temp:=Logger.s1;
ADDSTRING(ADR(tempRaw), ADR(temp), tempRawLen);

(* Sparo i COIL **)
FOR x:= 1 TO 65 DO
	temp:=CONCAT(SEL(MB_BitStatoCoil[x],'0','1'),';');
	ADDSTRING(ADR(tempRaw), ADR(temp), tempRawLen);
END_FOR

(* Sparo gli ingressi Digitali **)
FOR x:= 1 TO 358 DO
	temp:=CONCAT(SEL(MB_BitStato[x],'0','1'),';');
	ADDSTRING(ADR(tempRaw), ADR(temp), tempRawLen);
END_FOR

(* Sparo gli HOLDING **)
FOR x:= 1 TO 168 DO
	temp:=CONCAT(INT_TO_STRING(MB_RegistriHoldingLetti[x]),';');
	ADDSTRING(ADR(tempRaw), ADR(temp), tempRawLen);
END_FOR

(* Sparo gli integer **)
FOR x:= 1 TO 283 DO
	temp:=CONCAT(INT_TO_STRING(MB_RegistriLetti[x]),';');
	ADDSTRING(ADR(tempRaw), ADR(temp), tempRawLen);
END_FOR

	temp:=(INT_TO_STRING(MB_RegistriLetti[284]));
	ADDSTRING(ADR(tempRaw), ADR(temp), tempRawLen);

ADDSTRING(ADR(Logger.TData), ADR(tempRaw), Logger.TLen);
END_ACTION
ACTION Stm:
CASE state OF
	0:	(* Refresh time manager *)
		ReadTmr(IN:=NOT ReadTmr.Q);
		(*A tempo interrogo il nodo sempre che non ci sia qualcuno che lo sta interrogando in quel momento *)

		IF (ReadTmr.Q AND NodoDaInterrogareMB1=Address )OR Refresh_Now AND NOT InibiscoModbusMB1 THEN
			state := 10;
			ReadTmr.PT := T#10s;  (* moreno *)
			Refresh_Now := FALSE;
			InibiscoModbusMB1 := TRUE;
		END_IF

	(**** Leggo le Analogiche a Disposzione  ****)

	10:	(* richiedo lettura di tutti gli Input Register   *)

		Modbus.MB_Query.SlaveAddress := Address;
		Modbus.MB_Query.FunctionCode := 4;
		Read_StartAddress := 0 ;			(* richiedo lettura altri Parametri *)
		Read_Quantity := 20;
		ModBus.MB_Start := TRUE;
		state := 20;


	20:
		ModBus.MB_Query.Read_StartAddress := 0 ;			(* richiedo lettura altri Parametri *)
		ModBus.MB_Query.Read_Quantity := 20;
		ModBus.MB_Start := TRUE;
		Read_StartAddress := 0 ;
		state := 30;



	30:	(* Risposta all'interrogazione *)
		IF NOT ModBus.MB_Start   THEN
			VerificaFuctionCode:=ModBus.MB_Resp.FunctionCode;
			VerificaNodoLetto:=ModBus.MB_Resp.SlaveAddress;

			IF ModBus.MB_MASTER.MB_Error<>0 THEN
				state := 300;
			ELSE

				FOR x:= 0 TO ModBus.MB_Query.Read_Quantity DO
					MB_RegistriLetti[Read_StartAddress+x ] := ModBus.MB_Resp.Data[x];   	(* Vedi tabella *)
				END_FOR

			ModBus.MB_Query.Read_StartAddress := 20 ;			(* richiedo lettura altri Parametri *)
			ModBus.MB_Query.Read_Quantity := 20;
			ModBus.MB_Start := TRUE;
			Read_StartAddress := 20 ;
			state := 31;
			END_IF
		END_IF


	31:	(* Risposta all'interrogazione *)
		IF NOT ModBus.MB_Start   THEN
			VerificaFuctionCode:=ModBus.MB_Resp.FunctionCode;
			VerificaNodoLetto:=ModBus.MB_Resp.SlaveAddress;

			IF ModBus.MB_MASTER.MB_Error<>0 THEN
				state := 300;
			ELSE

				FOR x:= 0 TO ModBus.MB_Query.Read_Quantity DO
					MB_RegistriLetti[Read_StartAddress+x ] := ModBus.MB_Resp.Data[x];   	(* Vedi tabella *)
				END_FOR

			ModBus.MB_Query.Read_StartAddress := 40 ;			(* richiedo lettura altri Parametri *)
			ModBus.MB_Query.Read_Quantity := 20;
			ModBus.MB_Start := TRUE;
			Read_StartAddress := 40 ;
			state := 32;
			END_IF
		END_IF



	32:	(* Risposta all'interrogazione *)
		IF NOT ModBus.MB_Start   THEN
			VerificaFuctionCode:=ModBus.MB_Resp.FunctionCode;
			VerificaNodoLetto:=ModBus.MB_Resp.SlaveAddress;

			IF ModBus.MB_MASTER.MB_Error<>0 THEN
				state := 300;
			ELSE

				FOR x:= 0 TO ModBus.MB_Query.Read_Quantity DO
					MB_RegistriLetti[Read_StartAddress+x ] := ModBus.MB_Resp.Data[x];   	(* Vedi tabella *)
				END_FOR

			ModBus.MB_Query.Read_StartAddress := 60 ;			(* richiedo lettura altri Parametri *)
			ModBus.MB_Query.Read_Quantity := 20;
			ModBus.MB_Start := TRUE;
			Read_StartAddress := 60 ;
			state := 33;
			END_IF
		END_IF

	33:	(* Risposta all'interrogazione *)
		IF NOT ModBus.MB_Start   THEN
			VerificaFuctionCode:=ModBus.MB_Resp.FunctionCode;
			VerificaNodoLetto:=ModBus.MB_Resp.SlaveAddress;

			IF ModBus.MB_MASTER.MB_Error<>0 THEN
				state := 300;
			ELSE

				FOR x:= 0 TO ModBus.MB_Query.Read_Quantity DO
					MB_RegistriLetti[Read_StartAddress+x ] := ModBus.MB_Resp.Data[x];   	(* Vedi tabella *)
				END_FOR

			ModBus.MB_Query.Read_StartAddress := 80 ;			(* richiedo lettura altri Parametri *)
			ModBus.MB_Query.Read_Quantity := 20;
			ModBus.MB_Start := TRUE;
			Read_StartAddress := 80 ;
			state := 34;
			END_IF
		END_IF


	34:	(* Risposta all'interrogazione *)
		IF NOT ModBus.MB_Start   THEN
			VerificaFuctionCode:=ModBus.MB_Resp.FunctionCode;
			VerificaNodoLetto:=ModBus.MB_Resp.SlaveAddress;

			IF ModBus.MB_MASTER.MB_Error<>0 THEN
				state := 300;
			ELSE

				FOR x:= 0 TO ModBus.MB_Query.Read_Quantity DO
					MB_RegistriLetti[Read_StartAddress+x ] := ModBus.MB_Resp.Data[x];   	(* Vedi tabella *)
				END_FOR

			ModBus.MB_Query.Read_StartAddress := 100 ;			(* richiedo lettura altri Parametri *)
			ModBus.MB_Query.Read_Quantity := 20;
			ModBus.MB_Start := TRUE;
			Read_StartAddress := 100 ;
			state := 35;
			END_IF
		END_IF


	35:	(* Risposta all'interrogazione *)
		IF NOT ModBus.MB_Start   THEN
			VerificaFuctionCode:=ModBus.MB_Resp.FunctionCode;
			VerificaNodoLetto:=ModBus.MB_Resp.SlaveAddress;

			IF ModBus.MB_MASTER.MB_Error<>0 THEN
				state := 300;
			ELSE

				FOR x:= 0 TO ModBus.MB_Query.Read_Quantity DO
					MB_RegistriLetti[Read_StartAddress+x ] := ModBus.MB_Resp.Data[x];   	(* Vedi tabella *)
				END_FOR

			ModBus.MB_Query.Read_StartAddress := 120 ;			(* richiedo lettura altri Parametri *)
			ModBus.MB_Query.Read_Quantity := 20;
			ModBus.MB_Start := TRUE;
			Read_StartAddress := 120 ;
			state := 36;
			END_IF
		END_IF

	36:	(* Risposta all'interrogazione *)
		IF NOT ModBus.MB_Start   THEN
			VerificaFuctionCode:=ModBus.MB_Resp.FunctionCode;
			VerificaNodoLetto:=ModBus.MB_Resp.SlaveAddress;

			IF ModBus.MB_MASTER.MB_Error<>0 THEN
				state := 300;
			ELSE

				FOR x:= 0 TO ModBus.MB_Query.Read_Quantity DO
					MB_RegistriLetti[Read_StartAddress+x ] := ModBus.MB_Resp.Data[x];   	(* Vedi tabella *)
				END_FOR

			ModBus.MB_Query.Read_StartAddress := 140 ;			(* richiedo lettura altri Parametri *)
			ModBus.MB_Query.Read_Quantity := 20;
			ModBus.MB_Start := TRUE;
			Read_StartAddress := 140 ;
			state := 37;
			END_IF
		END_IF

	37:	(* Risposta all'interrogazione *)
		IF NOT ModBus.MB_Start   THEN
			VerificaFuctionCode:=ModBus.MB_Resp.FunctionCode;
			VerificaNodoLetto:=ModBus.MB_Resp.SlaveAddress;

			IF ModBus.MB_MASTER.MB_Error<>0 THEN
				state := 300;
			ELSE

				FOR x:= 0 TO ModBus.MB_Query.Read_Quantity DO
					MB_RegistriLetti[Read_StartAddress+x ] := ModBus.MB_Resp.Data[x];   	(* Vedi tabella *)
				END_FOR

			ModBus.MB_Query.Read_StartAddress := 160 ;			(* richiedo lettura altri Parametri *)
			ModBus.MB_Query.Read_Quantity := 20;
			ModBus.MB_Start := TRUE;
			Read_StartAddress := 160 ;
			state := 38;
			END_IF
		END_IF

	38:	(* Risposta all'interrogazione *)
		IF NOT ModBus.MB_Start   THEN
			VerificaFuctionCode:=ModBus.MB_Resp.FunctionCode;
			VerificaNodoLetto:=ModBus.MB_Resp.SlaveAddress;

			IF ModBus.MB_MASTER.MB_Error<>0 THEN
				state := 300;
			ELSE

				FOR x:= 0 TO ModBus.MB_Query.Read_Quantity DO
					MB_RegistriLetti[Read_StartAddress+x ] := ModBus.MB_Resp.Data[x];   	(* Vedi tabella *)
				END_FOR

			ModBus.MB_Query.Read_StartAddress := 180 ;			(* richiedo lettura altri Parametri *)
			ModBus.MB_Query.Read_Quantity := 20;
			ModBus.MB_Start := TRUE;
			Read_StartAddress := 180 ;
			state := 39;
			END_IF
		END_IF

	39:	(* Risposta all'interrogazione *)
		IF NOT ModBus.MB_Start   THEN
			VerificaFuctionCode:=ModBus.MB_Resp.FunctionCode;
			VerificaNodoLetto:=ModBus.MB_Resp.SlaveAddress;

			IF ModBus.MB_MASTER.MB_Error<>0 THEN
				state := 300;
			ELSE

				FOR x:= 0 TO ModBus.MB_Query.Read_Quantity DO
					MB_RegistriLetti[Read_StartAddress+x ] := ModBus.MB_Resp.Data[x];   	(* Vedi tabella *)
				END_FOR

			ModBus.MB_Query.Read_StartAddress := 200 ;			(* richiedo lettura altri Parametri *)
			ModBus.MB_Query.Read_Quantity := 20;
			ModBus.MB_Start := TRUE;
			Read_StartAddress := 200 ;
			state := 40;
			END_IF
		END_IF

	40:	(* Risposta all'interrogazione *)
		IF NOT ModBus.MB_Start   THEN
			VerificaFuctionCode:=ModBus.MB_Resp.FunctionCode;
			VerificaNodoLetto:=ModBus.MB_Resp.SlaveAddress;

			IF ModBus.MB_MASTER.MB_Error<>0 THEN
				state := 300;
			ELSE

				FOR x:= 0 TO ModBus.MB_Query.Read_Quantity DO
					MB_RegistriLetti[Read_StartAddress+x ] := ModBus.MB_Resp.Data[x];   	(* Vedi tabella *)
				END_FOR

			ModBus.MB_Query.Read_StartAddress := 220 ;			(* richiedo lettura altri Parametri *)
			ModBus.MB_Query.Read_Quantity := 20;
			ModBus.MB_Start := TRUE;
			Read_StartAddress := 220 ;
			state := 41;
			END_IF
		END_IF

	41:	(* Risposta all'interrogazione *)
		IF NOT ModBus.MB_Start   THEN
			VerificaFuctionCode:=ModBus.MB_Resp.FunctionCode;
			VerificaNodoLetto:=ModBus.MB_Resp.SlaveAddress;

			IF ModBus.MB_MASTER.MB_Error<>0 THEN
				state := 300;
			ELSE

				FOR x:= 0 TO ModBus.MB_Query.Read_Quantity DO
					MB_RegistriLetti[Read_StartAddress+x ] := ModBus.MB_Resp.Data[x];   	(* Vedi tabella *)
				END_FOR

			ModBus.MB_Query.Read_StartAddress := 240 ;			(* richiedo lettura altri Parametri *)
			ModBus.MB_Query.Read_Quantity := 20;
			ModBus.MB_Start := TRUE;
			Read_StartAddress := 240 ;
			state := 42;
			END_IF
		END_IF

	42:	(* Risposta all'interrogazione *)
		IF NOT ModBus.MB_Start   THEN
			VerificaFuctionCode:=ModBus.MB_Resp.FunctionCode;
			VerificaNodoLetto:=ModBus.MB_Resp.SlaveAddress;

			IF ModBus.MB_MASTER.MB_Error<>0 THEN
				state := 300;
			ELSE

				FOR x:= 0 TO ModBus.MB_Query.Read_Quantity DO
					MB_RegistriLetti[Read_StartAddress+x ] := ModBus.MB_Resp.Data[x];   	(* Vedi tabella *)
				END_FOR

			ModBus.MB_Query.Read_StartAddress := 260 ;			(* richiedo lettura altri Parametri *)
			ModBus.MB_Query.Read_Quantity := 20;
			ModBus.MB_Start := TRUE;
			Read_StartAddress := 260 ;
			state := 43;
			END_IF
		END_IF

	43:	(* Risposta all'interrogazione *)
		IF NOT ModBus.MB_Start   THEN
			VerificaFuctionCode:=ModBus.MB_Resp.FunctionCode;
			VerificaNodoLetto:=ModBus.MB_Resp.SlaveAddress;

			IF ModBus.MB_MASTER.MB_Error<>0 THEN
				state := 300;
			ELSE

				FOR x:= 0 TO ModBus.MB_Query.Read_Quantity DO
					MB_RegistriLetti[Read_StartAddress+x ] := ModBus.MB_Resp.Data[x];   	(* Vedi tabella *)
				END_FOR

			ModBus.MB_Query.Read_StartAddress := 280 ;			(* richiedo lettura altri Parametri *)
			ModBus.MB_Query.Read_Quantity := 4;
			ModBus.MB_Start := TRUE;
			Read_StartAddress := 280 ;
			state := 44;
			END_IF
		END_IF

	44:	(* Risposta all'interrogazione *)
		IF NOT ModBus.MB_Start   THEN
			VerificaFuctionCode:=ModBus.MB_Resp.FunctionCode;
			VerificaNodoLetto:=ModBus.MB_Resp.SlaveAddress;

			IF ModBus.MB_MASTER.MB_Error<>0 THEN
				state := 300;
			ELSE

				FOR x:= 0 TO ModBus.MB_Query.Read_Quantity DO
					MB_RegistriLetti[Read_StartAddress+x ] := ModBus.MB_Resp.Data[x];   	(* Vedi tabella *)
				END_FOR

		(*	ModBus.MB_Query.Read_StartAddress := 280 ;			(* richiedo lettura altri Parametri *)
			ModBus.MB_Query.Read_Quantity := 4;
			ModBus.MB_Start := TRUE;
			Read_StartAddress := 280 ; *)
			state := 50;
			END_IF
		END_IF





	50:	(* Risposta all'interrogazione Holding*)

		Modbus.MB_Query.FunctionCode := 3;
		Read_StartAddress := 0 ;			(* richiedo lettura altri Parametri *)
		Read_Quantity := 20;
		ModBus.MB_Start := TRUE;
		state := 51;

	51:	(* Risposta all'interrogazione *)
		IF NOT ModBus.MB_Start   THEN
			VerificaFuctionCode:=ModBus.MB_Resp.FunctionCode;
			VerificaNodoLetto:=ModBus.MB_Resp.SlaveAddress;

			IF ModBus.MB_MASTER.MB_Error<>0 THEN
				state := 300;
			ELSE

				FOR x:= 0 TO ModBus.MB_Query.Read_Quantity DO
					MB_RegistriHoldingLetti[Read_StartAddress+x ] := ModBus.MB_Resp.Data[x];   	(* Vedi tabella *)
				END_FOR

			ModBus.MB_Query.Read_StartAddress := 0 ;			(* richiedo lettura altri Parametri *)
			ModBus.MB_Query.Read_Quantity := 20;
			ModBus.MB_Start := TRUE;
			Read_StartAddress := 0 ;
			state := 511;
			END_IF
		END_IF


	511:	(* Risposta all'interrogazione *)
		IF NOT ModBus.MB_Start   THEN
			VerificaFuctionCode:=ModBus.MB_Resp.FunctionCode;
			VerificaNodoLetto:=ModBus.MB_Resp.SlaveAddress;

			IF ModBus.MB_MASTER.MB_Error<>0 THEN
				state := 300;
			ELSE

				FOR x:= 0 TO ModBus.MB_Query.Read_Quantity DO
					MB_RegistriHoldingLetti[Read_StartAddress+x ] := ModBus.MB_Resp.Data[x];   	(* Vedi tabella *)
				END_FOR

			ModBus.MB_Query.Read_StartAddress := 20 ;			(* richiedo lettura altri Parametri *)
			ModBus.MB_Query.Read_Quantity := 20;
			ModBus.MB_Start := TRUE;
			Read_StartAddress := 20 ;
			state := 52;
			END_IF
		END_IF

	52:	(* Risposta all'interrogazione *)
		IF NOT ModBus.MB_Start   THEN
			VerificaFuctionCode:=ModBus.MB_Resp.FunctionCode;
			VerificaNodoLetto:=ModBus.MB_Resp.SlaveAddress;

			IF ModBus.MB_MASTER.MB_Error<>0 THEN
				state := 300;
			ELSE

				FOR x:= 0 TO ModBus.MB_Query.Read_Quantity DO
					MB_RegistriHoldingLetti[Read_StartAddress+x ] := ModBus.MB_Resp.Data[x];   	(* Vedi tabella *)
				END_FOR

			ModBus.MB_Query.Read_StartAddress := 40 ;			(* richiedo lettura altri Parametri *)
			ModBus.MB_Query.Read_Quantity := 20;
			ModBus.MB_Start := TRUE;
			Read_StartAddress := 40 ;
			state := 53;
			END_IF
		END_IF

	53:	(* Risposta all'interrogazione *)
		IF NOT ModBus.MB_Start   THEN
			VerificaFuctionCode:=ModBus.MB_Resp.FunctionCode;
			VerificaNodoLetto:=ModBus.MB_Resp.SlaveAddress;

			IF ModBus.MB_MASTER.MB_Error<>0 THEN
				state := 300;
			ELSE

				FOR x:= 0 TO ModBus.MB_Query.Read_Quantity DO
					MB_RegistriHoldingLetti[Read_StartAddress+x ] := ModBus.MB_Resp.Data[x];   	(* Vedi tabella *)
				END_FOR

			ModBus.MB_Query.Read_StartAddress := 60 ;			(* richiedo lettura altri Parametri *)
			ModBus.MB_Query.Read_Quantity := 20;
			ModBus.MB_Start := TRUE;
			Read_StartAddress := 60 ;
			state := 54;
			END_IF
		END_IF

	54:	(* Risposta all'interrogazione *)
		IF NOT ModBus.MB_Start   THEN
			VerificaFuctionCode:=ModBus.MB_Resp.FunctionCode;
			VerificaNodoLetto:=ModBus.MB_Resp.SlaveAddress;

			IF ModBus.MB_MASTER.MB_Error<>0 THEN
				state := 300;
			ELSE

				FOR x:= 0 TO ModBus.MB_Query.Read_Quantity DO
					MB_RegistriHoldingLetti[Read_StartAddress+x ] := ModBus.MB_Resp.Data[x];   	(* Vedi tabella *)
				END_FOR

			ModBus.MB_Query.Read_StartAddress := 80 ;			(* richiedo lettura altri Parametri *)
			ModBus.MB_Query.Read_Quantity := 20;
			ModBus.MB_Start := TRUE;
			Read_StartAddress := 80 ;
			state := 55;
			END_IF
		END_IF

	55:	(* Risposta all'interrogazione *)
		IF NOT ModBus.MB_Start   THEN
			VerificaFuctionCode:=ModBus.MB_Resp.FunctionCode;
			VerificaNodoLetto:=ModBus.MB_Resp.SlaveAddress;

			IF ModBus.MB_MASTER.MB_Error<>0 THEN
				state := 300;
			ELSE

				FOR x:= 0 TO ModBus.MB_Query.Read_Quantity DO
					MB_RegistriHoldingLetti[Read_StartAddress+x ] := ModBus.MB_Resp.Data[x];   	(* Vedi tabella *)
				END_FOR

			ModBus.MB_Query.Read_StartAddress := 100 ;			(* richiedo lettura altri Parametri *)
			ModBus.MB_Query.Read_Quantity := 20;
			ModBus.MB_Start := TRUE;
			Read_StartAddress := 100 ;
			state := 56;
			END_IF
		END_IF

	56:	(* Risposta all'interrogazione *)
		IF NOT ModBus.MB_Start   THEN
			VerificaFuctionCode:=ModBus.MB_Resp.FunctionCode;
			VerificaNodoLetto:=ModBus.MB_Resp.SlaveAddress;

			IF ModBus.MB_MASTER.MB_Error<>0 THEN
				state := 300;
			ELSE

				FOR x:= 0 TO ModBus.MB_Query.Read_Quantity DO
					MB_RegistriHoldingLetti[Read_StartAddress+x ] := ModBus.MB_Resp.Data[x];   	(* Vedi tabella *)
				END_FOR

			ModBus.MB_Query.Read_StartAddress := 120 ;			(* richiedo lettura altri Parametri *)
			ModBus.MB_Query.Read_Quantity := 20;
			ModBus.MB_Start := TRUE;
			Read_StartAddress := 120 ;
			state := 57;
			END_IF
		END_IF

	57:	(* Risposta all'interrogazione *)
		IF NOT ModBus.MB_Start   THEN
			VerificaFuctionCode:=ModBus.MB_Resp.FunctionCode;
			VerificaNodoLetto:=ModBus.MB_Resp.SlaveAddress;

			IF ModBus.MB_MASTER.MB_Error<>0 THEN
				state := 300;
			ELSE

				FOR x:= 0 TO ModBus.MB_Query.Read_Quantity DO
					MB_RegistriHoldingLetti[Read_StartAddress+x ] := ModBus.MB_Resp.Data[x];   	(* Vedi tabella *)
				END_FOR

			ModBus.MB_Query.Read_StartAddress := 140 ;			(* richiedo lettura altri Parametri *)
			ModBus.MB_Query.Read_Quantity := 20;
			ModBus.MB_Start := TRUE;
			Read_StartAddress := 140 ;
			state := 58;
			END_IF
		END_IF

	58:	(* Risposta all'interrogazione *)
		IF NOT ModBus.MB_Start   THEN
			VerificaFuctionCode:=ModBus.MB_Resp.FunctionCode;
			VerificaNodoLetto:=ModBus.MB_Resp.SlaveAddress;

			IF ModBus.MB_MASTER.MB_Error<>0 THEN
				state := 300;
			ELSE

				FOR x:= 0 TO ModBus.MB_Query.Read_Quantity DO
					MB_RegistriHoldingLetti[Read_StartAddress+x ] := ModBus.MB_Resp.Data[x];   	(* Vedi tabella *)
				END_FOR

			ModBus.MB_Query.Read_StartAddress := 160 ;			(* richiedo lettura altri Parametri *)
			ModBus.MB_Query.Read_Quantity := 8;
			ModBus.MB_Start := TRUE;
			Read_StartAddress := 160 ;
			state := 59;
			END_IF
		END_IF

	59:	(* Risposta all'interrogazione *)
		IF NOT ModBus.MB_Start   THEN
			VerificaFuctionCode:=ModBus.MB_Resp.FunctionCode;
			VerificaNodoLetto:=ModBus.MB_Resp.SlaveAddress;

			IF ModBus.MB_MASTER.MB_Error<>0 THEN
				state := 300;
			ELSE

				FOR x:= 0 TO ModBus.MB_Query.Read_Quantity DO
					MB_RegistriHoldingLetti[Read_StartAddress+x ] := ModBus.MB_Resp.Data[x];   	(* Vedi tabella *)
				END_FOR

		(*	ModBus.MB_Query.Read_StartAddress := 160 ;			(* richiedo lettura altri Parametri *)
			ModBus.MB_Query.Read_Quantity := 20;
			ModBus.MB_Start := TRUE;
			Read_StartAddress := 160 ; *)
			state := 100;
			END_IF
		END_IF





	100: (* Rispota Altri paramenti Digital Input *)
		IF NOT ModBus.MB_Start  THEN

			IF ModBus.MB_MASTER.MB_Error<>0 THEN
				state := 300;
			ELSE
				Modbus.MB_Query.SlaveAddress := Address;
				Modbus.MB_Query.FunctionCode := 2;
				ModBus.MB_Query.Read_StartAddress := 0;	(* richiedo lettura altri Parametri *)
				ModBus.MB_Query.Read_Quantity := 64;
				ModBus.MB_Start := TRUE;

				state:=105;
			END_IF
		END_IF
	105: (* Rispota Altri paramenti *)

		IF NOT ModBus.MB_Start  THEN

			IF ModBus.MB_MASTER.MB_Error<>0 THEN
				state := 300;
			ELSE

				MB_BitStato[0]:=ModBus.MB_MASTER.ReceiveBuffer.Data[3].0; (*Vedi Tabella *)
				MB_BitStato[1]:=ModBus.MB_MASTER.ReceiveBuffer.Data[3].1; (*Vedi Tabella *)
				MB_BitStato[2]:=ModBus.MB_MASTER.ReceiveBuffer.Data[3].2; (*Vedi Tabella *)
				MB_BitStato[3]:=ModBus.MB_MASTER.ReceiveBuffer.Data[3].3; (*Vedi Tabella *)
				MB_BitStato[4]:=ModBus.MB_MASTER.ReceiveBuffer.Data[3].4; (*Vedi Tabella *)
				MB_BitStato[5]:=ModBus.MB_MASTER.ReceiveBuffer.Data[3].5; (*Vedi Tabella *)
				MB_BitStato[6]:=ModBus.MB_MASTER.ReceiveBuffer.Data[3].6; (*Vedi Tabella *)
				MB_BitStato[7]:=ModBus.MB_MASTER.ReceiveBuffer.Data[3].7; (*Vedi Tabella *)
				MB_BitStato[8]:=ModBus.MB_MASTER.ReceiveBuffer.Data[4].0; (*Vedi Tabella *)
				MB_BitStato[9]:=ModBus.MB_MASTER.ReceiveBuffer.Data[4].1; (*Vedi Tabella *)
				MB_BitStato[10]:=ModBus.MB_MASTER.ReceiveBuffer.Data[4].2; (*Vedi Tabella *)
				MB_BitStato[11]:=ModBus.MB_MASTER.ReceiveBuffer.Data[4].3; (*Vedi Tabella *)
				MB_BitStato[12]:=ModBus.MB_MASTER.ReceiveBuffer.Data[4].4; (*Vedi Tabella *)
				MB_BitStato[13]:=ModBus.MB_MASTER.ReceiveBuffer.Data[4].5; (*Vedi Tabella *)
				MB_BitStato[14]:=ModBus.MB_MASTER.ReceiveBuffer.Data[4].6; (*Vedi Tabella *)
				MB_BitStato[15]:=ModBus.MB_MASTER.ReceiveBuffer.Data[4].7; (*Vedi Tabella *)
				MB_BitStato[16]:=ModBus.MB_MASTER.ReceiveBuffer.Data[5].0; (*Vedi Tabella *)
				MB_BitStato[17]:=ModBus.MB_MASTER.ReceiveBuffer.Data[5].1; (*Vedi Tabella *)
				MB_BitStato[18]:=ModBus.MB_MASTER.ReceiveBuffer.Data[5].2; (*Vedi Tabella *)
				MB_BitStato[19]:=ModBus.MB_MASTER.ReceiveBuffer.Data[5].3; (*Vedi Tabella *)
				MB_BitStato[20]:=ModBus.MB_MASTER.ReceiveBuffer.Data[5].4; (*Vedi Tabella *)
				MB_BitStato[21]:=ModBus.MB_MASTER.ReceiveBuffer.Data[5].5; (*Vedi Tabella *)
				MB_BitStato[22]:=ModBus.MB_MASTER.ReceiveBuffer.Data[5].6; (*Vedi Tabella *)
				MB_BitStato[23]:=ModBus.MB_MASTER.ReceiveBuffer.Data[5].7; (*Vedi Tabella *)
				MB_BitStato[24]:=ModBus.MB_MASTER.ReceiveBuffer.Data[6].0; (*Vedi Tabella *)
				MB_BitStato[25]:=ModBus.MB_MASTER.ReceiveBuffer.Data[6].1; (*Vedi Tabella *)
				MB_BitStato[26]:=ModBus.MB_MASTER.ReceiveBuffer.Data[6].2; (*Vedi Tabella *)
				MB_BitStato[27]:=ModBus.MB_MASTER.ReceiveBuffer.Data[6].3; (*Vedi Tabella *)
				MB_BitStato[28]:=ModBus.MB_MASTER.ReceiveBuffer.Data[6].4; (*Vedi Tabella *)
				MB_BitStato[29]:=ModBus.MB_MASTER.ReceiveBuffer.Data[6].5; (*Vedi Tabella *)
				MB_BitStato[30]:=ModBus.MB_MASTER.ReceiveBuffer.Data[6].6; (*Vedi Tabella *)
				MB_BitStato[31]:=ModBus.MB_MASTER.ReceiveBuffer.Data[6].7; (*Vedi Tabella *)
				MB_BitStato[32]:=ModBus.MB_MASTER.ReceiveBuffer.Data[7].0; (*Vedi Tabella *)
				MB_BitStato[33]:=ModBus.MB_MASTER.ReceiveBuffer.Data[7].1; (*Vedi Tabella *)
				MB_BitStato[34]:=ModBus.MB_MASTER.ReceiveBuffer.Data[7].2; (*Vedi Tabella *)
				MB_BitStato[35]:=ModBus.MB_MASTER.ReceiveBuffer.Data[7].3; (*Vedi Tabella *)
				MB_BitStato[36]:=ModBus.MB_MASTER.ReceiveBuffer.Data[7].4; (*Vedi Tabella *)
				MB_BitStato[37]:=ModBus.MB_MASTER.ReceiveBuffer.Data[7].5; (*Vedi Tabella *)
				MB_BitStato[38]:=ModBus.MB_MASTER.ReceiveBuffer.Data[7].6; (*Vedi Tabella *)
				MB_BitStato[39]:=ModBus.MB_MASTER.ReceiveBuffer.Data[7].7; (*Vedi Tabella *)
				MB_BitStato[40]:=ModBus.MB_MASTER.ReceiveBuffer.Data[8].0; (*Vedi Tabella *)
				MB_BitStato[41]:=ModBus.MB_MASTER.ReceiveBuffer.Data[8].1; (*Vedi Tabella *)
				MB_BitStato[42]:=ModBus.MB_MASTER.ReceiveBuffer.Data[8].2; (*Vedi Tabella *)
				MB_BitStato[43]:=ModBus.MB_MASTER.ReceiveBuffer.Data[8].3; (*Vedi Tabella *)
				MB_BitStato[44]:=ModBus.MB_MASTER.ReceiveBuffer.Data[8].4; (*Vedi Tabella *)
				MB_BitStato[45]:=ModBus.MB_MASTER.ReceiveBuffer.Data[8].5; (*Vedi Tabella *)
				MB_BitStato[46]:=ModBus.MB_MASTER.ReceiveBuffer.Data[8].6; (*Vedi Tabella *)
				MB_BitStato[47]:=ModBus.MB_MASTER.ReceiveBuffer.Data[8].7; (*Vedi Tabella *)
				MB_BitStato[48]:=ModBus.MB_MASTER.ReceiveBuffer.Data[9].0; (*Vedi Tabella *)
				MB_BitStato[49]:=ModBus.MB_MASTER.ReceiveBuffer.Data[9].1; (*Vedi Tabella *)
				MB_BitStato[50]:=ModBus.MB_MASTER.ReceiveBuffer.Data[9].2; (*Vedi Tabella *)
				MB_BitStato[51]:=ModBus.MB_MASTER.ReceiveBuffer.Data[9].3; (*Vedi Tabella *)
				MB_BitStato[52]:=ModBus.MB_MASTER.ReceiveBuffer.Data[9].4; (*Vedi Tabella *)
				MB_BitStato[53]:=ModBus.MB_MASTER.ReceiveBuffer.Data[9].5; (*Vedi Tabella *)
				MB_BitStato[54]:=ModBus.MB_MASTER.ReceiveBuffer.Data[9].6; (*Vedi Tabella *)
				MB_BitStato[55]:=ModBus.MB_MASTER.ReceiveBuffer.Data[9].7; (*Vedi Tabella *)
				MB_BitStato[56]:=ModBus.MB_MASTER.ReceiveBuffer.Data[10].0; (*Vedi Tabella *)
				MB_BitStato[57]:=ModBus.MB_MASTER.ReceiveBuffer.Data[10].1; (*Vedi Tabella *)
				MB_BitStato[58]:=ModBus.MB_MASTER.ReceiveBuffer.Data[10].2; (*Vedi Tabella *)
				MB_BitStato[59]:=ModBus.MB_MASTER.ReceiveBuffer.Data[10].3; (*Vedi Tabella *)
				MB_BitStato[60]:=ModBus.MB_MASTER.ReceiveBuffer.Data[10].4; (*Vedi Tabella *)
				MB_BitStato[61]:=ModBus.MB_MASTER.ReceiveBuffer.Data[10].5; (*Vedi Tabella *)
				MB_BitStato[62]:=ModBus.MB_MASTER.ReceiveBuffer.Data[10].6; (*Vedi Tabella *)
				MB_BitStato[63]:=ModBus.MB_MASTER.ReceiveBuffer.Data[10].7; (*Vedi Tabella *)

				state:=110;

			END_IF
		END_IF

	110: (* Rispota Altri paramenti *)
		IF NOT ModBus.MB_Start  THEN

			IF ModBus.MB_MASTER.MB_Error<>0 THEN
				state := 300;
			ELSE
				Modbus.MB_Query.SlaveAddress := Address;
				Modbus.MB_Query.FunctionCode := 2;
				ModBus.MB_Query.Read_StartAddress := 64;
				ModBus.MB_Query.Read_Quantity := 64;
				ModBus.MB_Start := TRUE;

				state:=115;
			END_IF
		END_IF
	115: (* Rispota Altri paramenti *)

		IF NOT ModBus.MB_Start  THEN

			IF ModBus.MB_MASTER.MB_Error<>0 THEN
				state := 300;
			ELSE

				MB_BitStato[64]:=ModBus.MB_MASTER.ReceiveBuffer.Data[3].0; (*Vedi Tabella *)
				MB_BitStato[65]:=ModBus.MB_MASTER.ReceiveBuffer.Data[3].1; (*Vedi Tabella *)
				MB_BitStato[66]:=ModBus.MB_MASTER.ReceiveBuffer.Data[3].2; (*Vedi Tabella *)
				MB_BitStato[67]:=ModBus.MB_MASTER.ReceiveBuffer.Data[3].3; (*Vedi Tabella *)
				MB_BitStato[68]:=ModBus.MB_MASTER.ReceiveBuffer.Data[3].4; (*Vedi Tabella *)
				MB_BitStato[69]:=ModBus.MB_MASTER.ReceiveBuffer.Data[3].5; (*Vedi Tabella *)
				MB_BitStato[70]:=ModBus.MB_MASTER.ReceiveBuffer.Data[3].6; (*Vedi Tabella *)
				MB_BitStato[71]:=ModBus.MB_MASTER.ReceiveBuffer.Data[3].7; (*Vedi Tabella *)
				MB_BitStato[72]:=ModBus.MB_MASTER.ReceiveBuffer.Data[4].0; (*Vedi Tabella *)
				MB_BitStato[73]:=ModBus.MB_MASTER.ReceiveBuffer.Data[4].1; (*Vedi Tabella *)
				MB_BitStato[74]:=ModBus.MB_MASTER.ReceiveBuffer.Data[4].2; (*Vedi Tabella *)
				MB_BitStato[75]:=ModBus.MB_MASTER.ReceiveBuffer.Data[4].3; (*Vedi Tabella *)
				MB_BitStato[76]:=ModBus.MB_MASTER.ReceiveBuffer.Data[4].4; (*Vedi Tabella *)
				MB_BitStato[77]:=ModBus.MB_MASTER.ReceiveBuffer.Data[4].5; (*Vedi Tabella *)
				MB_BitStato[78]:=ModBus.MB_MASTER.ReceiveBuffer.Data[4].6; (*Vedi Tabella *)
				MB_BitStato[79]:=ModBus.MB_MASTER.ReceiveBuffer.Data[4].7; (*Vedi Tabella *)
				MB_BitStato[80]:=ModBus.MB_MASTER.ReceiveBuffer.Data[5].0; (*Vedi Tabella *)
				MB_BitStato[81]:=ModBus.MB_MASTER.ReceiveBuffer.Data[5].1; (*Vedi Tabella *)
				MB_BitStato[82]:=ModBus.MB_MASTER.ReceiveBuffer.Data[5].2; (*Vedi Tabella *)
				MB_BitStato[83]:=ModBus.MB_MASTER.ReceiveBuffer.Data[5].3; (*Vedi Tabella *)
				MB_BitStato[84]:=ModBus.MB_MASTER.ReceiveBuffer.Data[5].4; (*Vedi Tabella *)
				MB_BitStato[85]:=ModBus.MB_MASTER.ReceiveBuffer.Data[5].5; (*Vedi Tabella *)
				MB_BitStato[86]:=ModBus.MB_MASTER.ReceiveBuffer.Data[5].6; (*Vedi Tabella *)
				MB_BitStato[87]:=ModBus.MB_MASTER.ReceiveBuffer.Data[5].7; (*Vedi Tabella *)
				MB_BitStato[88]:=ModBus.MB_MASTER.ReceiveBuffer.Data[6].0; (*Vedi Tabella *)
				MB_BitStato[89]:=ModBus.MB_MASTER.ReceiveBuffer.Data[6].1; (*Vedi Tabella *)
				MB_BitStato[90]:=ModBus.MB_MASTER.ReceiveBuffer.Data[6].2; (*Vedi Tabella *)
				MB_BitStato[91]:=ModBus.MB_MASTER.ReceiveBuffer.Data[6].3; (*Vedi Tabella *)
				MB_BitStato[92]:=ModBus.MB_MASTER.ReceiveBuffer.Data[6].4; (*Vedi Tabella *)
				MB_BitStato[93]:=ModBus.MB_MASTER.ReceiveBuffer.Data[6].5; (*Vedi Tabella *)
				MB_BitStato[94]:=ModBus.MB_MASTER.ReceiveBuffer.Data[6].6; (*Vedi Tabella *)
				MB_BitStato[95]:=ModBus.MB_MASTER.ReceiveBuffer.Data[6].7; (*Vedi Tabella *)
				MB_BitStato[96]:=ModBus.MB_MASTER.ReceiveBuffer.Data[7].0; (*Vedi Tabella *)
				MB_BitStato[97]:=ModBus.MB_MASTER.ReceiveBuffer.Data[7].1; (*Vedi Tabella *)
				MB_BitStato[98]:=ModBus.MB_MASTER.ReceiveBuffer.Data[7].2; (*Vedi Tabella *)
				MB_BitStato[99]:=ModBus.MB_MASTER.ReceiveBuffer.Data[7].3; (*Vedi Tabella *)
				MB_BitStato[100]:=ModBus.MB_MASTER.ReceiveBuffer.Data[7].4; (*Vedi Tabella *)
				MB_BitStato[101]:=ModBus.MB_MASTER.ReceiveBuffer.Data[7].5; (*Vedi Tabella *)
				MB_BitStato[102]:=ModBus.MB_MASTER.ReceiveBuffer.Data[7].6; (*Vedi Tabella *)
				MB_BitStato[103]:=ModBus.MB_MASTER.ReceiveBuffer.Data[7].7; (*Vedi Tabella *)
				MB_BitStato[104]:=ModBus.MB_MASTER.ReceiveBuffer.Data[8].0; (*Vedi Tabella *)
				MB_BitStato[105]:=ModBus.MB_MASTER.ReceiveBuffer.Data[8].1; (*Vedi Tabella *)
				MB_BitStato[106]:=ModBus.MB_MASTER.ReceiveBuffer.Data[8].2; (*Vedi Tabella *)
				MB_BitStato[107]:=ModBus.MB_MASTER.ReceiveBuffer.Data[8].3; (*Vedi Tabella *)
				MB_BitStato[108]:=ModBus.MB_MASTER.ReceiveBuffer.Data[8].4; (*Vedi Tabella *)
				MB_BitStato[109]:=ModBus.MB_MASTER.ReceiveBuffer.Data[8].5; (*Vedi Tabella *)
				MB_BitStato[110]:=ModBus.MB_MASTER.ReceiveBuffer.Data[8].6; (*Vedi Tabella *)
				MB_BitStato[111]:=ModBus.MB_MASTER.ReceiveBuffer.Data[8].7; (*Vedi Tabella *)
				MB_BitStato[112]:=ModBus.MB_MASTER.ReceiveBuffer.Data[9].0; (*Vedi Tabella *)
				MB_BitStato[113]:=ModBus.MB_MASTER.ReceiveBuffer.Data[9].1; (*Vedi Tabella *)
				MB_BitStato[114]:=ModBus.MB_MASTER.ReceiveBuffer.Data[9].2; (*Vedi Tabella *)
				MB_BitStato[115]:=ModBus.MB_MASTER.ReceiveBuffer.Data[9].3; (*Vedi Tabella *)
				MB_BitStato[116]:=ModBus.MB_MASTER.ReceiveBuffer.Data[9].4; (*Vedi Tabella *)
				MB_BitStato[117]:=ModBus.MB_MASTER.ReceiveBuffer.Data[9].5; (*Vedi Tabella *)
				MB_BitStato[118]:=ModBus.MB_MASTER.ReceiveBuffer.Data[9].6; (*Vedi Tabella *)
				MB_BitStato[119]:=ModBus.MB_MASTER.ReceiveBuffer.Data[9].7; (*Vedi Tabella *)
				MB_BitStato[120]:=ModBus.MB_MASTER.ReceiveBuffer.Data[10].0; (*Vedi Tabella *)
				MB_BitStato[121]:=ModBus.MB_MASTER.ReceiveBuffer.Data[10].1; (*Vedi Tabella *)
				MB_BitStato[122]:=ModBus.MB_MASTER.ReceiveBuffer.Data[10].2; (*Vedi Tabella *)
				MB_BitStato[123]:=ModBus.MB_MASTER.ReceiveBuffer.Data[10].3; (*Vedi Tabella *)
				MB_BitStato[124]:=ModBus.MB_MASTER.ReceiveBuffer.Data[10].4; (*Vedi Tabella *)
				MB_BitStato[125]:=ModBus.MB_MASTER.ReceiveBuffer.Data[10].5; (*Vedi Tabella *)
				MB_BitStato[126]:=ModBus.MB_MASTER.ReceiveBuffer.Data[10].6; (*Vedi Tabella *)
				MB_BitStato[127]:=ModBus.MB_MASTER.ReceiveBuffer.Data[10].7; (*Vedi Tabella *)


				state:=120;

			END_IF
		END_IF


	120: (* Rispota Altri paramenti *)
		IF NOT ModBus.MB_Start  THEN

			IF ModBus.MB_MASTER.MB_Error<>0 THEN
				state := 300;
			ELSE
				Modbus.MB_Query.SlaveAddress := Address;
				Modbus.MB_Query.FunctionCode := 2;
				ModBus.MB_Query.Read_StartAddress := 128;
				ModBus.MB_Query.Read_Quantity := 64;
				ModBus.MB_Start := TRUE;

				state:=125;
			END_IF
		END_IF
	125: (* Rispota Altri paramenti *)

		IF NOT ModBus.MB_Start  THEN

			IF ModBus.MB_MASTER.MB_Error<>0 THEN
				state := 300;
			ELSE

				MB_BitStato[128]:=ModBus.MB_MASTER.ReceiveBuffer.Data[3].0; (*Vedi Tabella *)
				MB_BitStato[129]:=ModBus.MB_MASTER.ReceiveBuffer.Data[3].1; (*Vedi Tabella *)
				MB_BitStato[130]:=ModBus.MB_MASTER.ReceiveBuffer.Data[3].2; (*Vedi Tabella *)
				MB_BitStato[131]:=ModBus.MB_MASTER.ReceiveBuffer.Data[3].3; (*Vedi Tabella *)
				MB_BitStato[132]:=ModBus.MB_MASTER.ReceiveBuffer.Data[3].4; (*Vedi Tabella *)
				MB_BitStato[133]:=ModBus.MB_MASTER.ReceiveBuffer.Data[3].5; (*Vedi Tabella *)
				MB_BitStato[134]:=ModBus.MB_MASTER.ReceiveBuffer.Data[3].6; (*Vedi Tabella *)
				MB_BitStato[135]:=ModBus.MB_MASTER.ReceiveBuffer.Data[3].7; (*Vedi Tabella *)
				MB_BitStato[136]:=ModBus.MB_MASTER.ReceiveBuffer.Data[4].0; (*Vedi Tabella *)
				MB_BitStato[137]:=ModBus.MB_MASTER.ReceiveBuffer.Data[4].1; (*Vedi Tabella *)
				MB_BitStato[138]:=ModBus.MB_MASTER.ReceiveBuffer.Data[4].2; (*Vedi Tabella *)
				MB_BitStato[139]:=ModBus.MB_MASTER.ReceiveBuffer.Data[4].3; (*Vedi Tabella *)
				MB_BitStato[140]:=ModBus.MB_MASTER.ReceiveBuffer.Data[4].4; (*Vedi Tabella *)
				MB_BitStato[141]:=ModBus.MB_MASTER.ReceiveBuffer.Data[4].5; (*Vedi Tabella *)
				MB_BitStato[142]:=ModBus.MB_MASTER.ReceiveBuffer.Data[4].6; (*Vedi Tabella *)
				MB_BitStato[143]:=ModBus.MB_MASTER.ReceiveBuffer.Data[4].7; (*Vedi Tabella *)
				MB_BitStato[144]:=ModBus.MB_MASTER.ReceiveBuffer.Data[5].0; (*Vedi Tabella *)
				MB_BitStato[145]:=ModBus.MB_MASTER.ReceiveBuffer.Data[5].1; (*Vedi Tabella *)
				MB_BitStato[146]:=ModBus.MB_MASTER.ReceiveBuffer.Data[5].2; (*Vedi Tabella *)
				MB_BitStato[147]:=ModBus.MB_MASTER.ReceiveBuffer.Data[5].3; (*Vedi Tabella *)
				MB_BitStato[148]:=ModBus.MB_MASTER.ReceiveBuffer.Data[5].4; (*Vedi Tabella *)
				MB_BitStato[149]:=ModBus.MB_MASTER.ReceiveBuffer.Data[5].5; (*Vedi Tabella *)
				MB_BitStato[150]:=ModBus.MB_MASTER.ReceiveBuffer.Data[5].6; (*Vedi Tabella *)
				MB_BitStato[151]:=ModBus.MB_MASTER.ReceiveBuffer.Data[5].7; (*Vedi Tabella *)
				MB_BitStato[152]:=ModBus.MB_MASTER.ReceiveBuffer.Data[6].0; (*Vedi Tabella *)
				MB_BitStato[153]:=ModBus.MB_MASTER.ReceiveBuffer.Data[6].1; (*Vedi Tabella *)
				MB_BitStato[154]:=ModBus.MB_MASTER.ReceiveBuffer.Data[6].2; (*Vedi Tabella *)
				MB_BitStato[155]:=ModBus.MB_MASTER.ReceiveBuffer.Data[6].3; (*Vedi Tabella *)
				MB_BitStato[156]:=ModBus.MB_MASTER.ReceiveBuffer.Data[6].4; (*Vedi Tabella *)
				MB_BitStato[157]:=ModBus.MB_MASTER.ReceiveBuffer.Data[6].5; (*Vedi Tabella *)
				MB_BitStato[158]:=ModBus.MB_MASTER.ReceiveBuffer.Data[6].6; (*Vedi Tabella *)
				MB_BitStato[159]:=ModBus.MB_MASTER.ReceiveBuffer.Data[6].7; (*Vedi Tabella *)
				MB_BitStato[160]:=ModBus.MB_MASTER.ReceiveBuffer.Data[7].0; (*Vedi Tabella *)
				MB_BitStato[161]:=ModBus.MB_MASTER.ReceiveBuffer.Data[7].1; (*Vedi Tabella *)
				MB_BitStato[162]:=ModBus.MB_MASTER.ReceiveBuffer.Data[7].2; (*Vedi Tabella *)
				MB_BitStato[163]:=ModBus.MB_MASTER.ReceiveBuffer.Data[7].3; (*Vedi Tabella *)
				MB_BitStato[164]:=ModBus.MB_MASTER.ReceiveBuffer.Data[7].4; (*Vedi Tabella *)
				MB_BitStato[165]:=ModBus.MB_MASTER.ReceiveBuffer.Data[7].5; (*Vedi Tabella *)
				MB_BitStato[166]:=ModBus.MB_MASTER.ReceiveBuffer.Data[7].6; (*Vedi Tabella *)
				MB_BitStato[167]:=ModBus.MB_MASTER.ReceiveBuffer.Data[7].7; (*Vedi Tabella *)
				MB_BitStato[168]:=ModBus.MB_MASTER.ReceiveBuffer.Data[8].0; (*Vedi Tabella *)
				MB_BitStato[169]:=ModBus.MB_MASTER.ReceiveBuffer.Data[8].1; (*Vedi Tabella *)
				MB_BitStato[170]:=ModBus.MB_MASTER.ReceiveBuffer.Data[8].2; (*Vedi Tabella *)
				MB_BitStato[171]:=ModBus.MB_MASTER.ReceiveBuffer.Data[8].3; (*Vedi Tabella *)
				MB_BitStato[172]:=ModBus.MB_MASTER.ReceiveBuffer.Data[8].4; (*Vedi Tabella *)
				MB_BitStato[173]:=ModBus.MB_MASTER.ReceiveBuffer.Data[8].5; (*Vedi Tabella *)
				MB_BitStato[174]:=ModBus.MB_MASTER.ReceiveBuffer.Data[8].6; (*Vedi Tabella *)
				MB_BitStato[175]:=ModBus.MB_MASTER.ReceiveBuffer.Data[8].7; (*Vedi Tabella *)
				MB_BitStato[176]:=ModBus.MB_MASTER.ReceiveBuffer.Data[9].0; (*Vedi Tabella *)
				MB_BitStato[177]:=ModBus.MB_MASTER.ReceiveBuffer.Data[9].1; (*Vedi Tabella *)
				MB_BitStato[178]:=ModBus.MB_MASTER.ReceiveBuffer.Data[9].2; (*Vedi Tabella *)
				MB_BitStato[179]:=ModBus.MB_MASTER.ReceiveBuffer.Data[9].3; (*Vedi Tabella *)
				MB_BitStato[180]:=ModBus.MB_MASTER.ReceiveBuffer.Data[9].4; (*Vedi Tabella *)
				MB_BitStato[181]:=ModBus.MB_MASTER.ReceiveBuffer.Data[9].5; (*Vedi Tabella *)
				MB_BitStato[182]:=ModBus.MB_MASTER.ReceiveBuffer.Data[9].6; (*Vedi Tabella *)
				MB_BitStato[183]:=ModBus.MB_MASTER.ReceiveBuffer.Data[9].7; (*Vedi Tabella *)
				MB_BitStato[184]:=ModBus.MB_MASTER.ReceiveBuffer.Data[10].0; (*Vedi Tabella *)
				MB_BitStato[185]:=ModBus.MB_MASTER.ReceiveBuffer.Data[10].1; (*Vedi Tabella *)
				MB_BitStato[186]:=ModBus.MB_MASTER.ReceiveBuffer.Data[10].2; (*Vedi Tabella *)
				MB_BitStato[187]:=ModBus.MB_MASTER.ReceiveBuffer.Data[10].3; (*Vedi Tabella *)
				MB_BitStato[188]:=ModBus.MB_MASTER.ReceiveBuffer.Data[10].4; (*Vedi Tabella *)
				MB_BitStato[189]:=ModBus.MB_MASTER.ReceiveBuffer.Data[10].5; (*Vedi Tabella *)
				MB_BitStato[190]:=ModBus.MB_MASTER.ReceiveBuffer.Data[10].6; (*Vedi Tabella *)
				MB_BitStato[191]:=ModBus.MB_MASTER.ReceiveBuffer.Data[10].7; (*Vedi Tabella *)


				state:=130;

			END_IF
		END_IF


	130: (* Rispota Altri paramenti COIL *)
		IF NOT ModBus.MB_Start  THEN

			IF ModBus.MB_MASTER.MB_Error<>0 THEN
				state := 300;
			ELSE
				Modbus.MB_Query.SlaveAddress := Address;
				Modbus.MB_Query.FunctionCode := 2;
				ModBus.MB_Query.Read_StartAddress := 192;	(* richiedo lettura altri Parametri *)
				ModBus.MB_Query.Read_Quantity := 64;
				ModBus.MB_Start := TRUE;

				state:=135;
			END_IF
		END_IF
	135: (* Rispota Altri paramenti *)

		IF NOT ModBus.MB_Start  THEN

			IF ModBus.MB_MASTER.MB_Error<>0 THEN
				state := 300;
			ELSE

				MB_BitStato[192]:=ModBus.MB_MASTER.ReceiveBuffer.Data[3].0; (*Vedi Tabella *)
				MB_BitStato[193]:=ModBus.MB_MASTER.ReceiveBuffer.Data[3].1; (*Vedi Tabella *)
				MB_BitStato[194]:=ModBus.MB_MASTER.ReceiveBuffer.Data[3].2; (*Vedi Tabella *)
				MB_BitStato[195]:=ModBus.MB_MASTER.ReceiveBuffer.Data[3].3; (*Vedi Tabella *)
				MB_BitStato[196]:=ModBus.MB_MASTER.ReceiveBuffer.Data[3].4; (*Vedi Tabella *)
				MB_BitStato[197]:=ModBus.MB_MASTER.ReceiveBuffer.Data[3].5; (*Vedi Tabella *)
				MB_BitStato[198]:=ModBus.MB_MASTER.ReceiveBuffer.Data[3].6; (*Vedi Tabella *)
				MB_BitStato[199]:=ModBus.MB_MASTER.ReceiveBuffer.Data[3].7; (*Vedi Tabella *)
				MB_BitStato[200]:=ModBus.MB_MASTER.ReceiveBuffer.Data[4].0; (*Vedi Tabella *)
				MB_BitStato[201]:=ModBus.MB_MASTER.ReceiveBuffer.Data[4].1; (*Vedi Tabella *)
				MB_BitStato[202]:=ModBus.MB_MASTER.ReceiveBuffer.Data[4].2; (*Vedi Tabella *)
				MB_BitStato[203]:=ModBus.MB_MASTER.ReceiveBuffer.Data[4].3; (*Vedi Tabella *)
				MB_BitStato[204]:=ModBus.MB_MASTER.ReceiveBuffer.Data[4].4; (*Vedi Tabella *)
				MB_BitStato[205]:=ModBus.MB_MASTER.ReceiveBuffer.Data[4].5; (*Vedi Tabella *)
				MB_BitStato[206]:=ModBus.MB_MASTER.ReceiveBuffer.Data[4].6; (*Vedi Tabella *)
				MB_BitStato[207]:=ModBus.MB_MASTER.ReceiveBuffer.Data[4].7; (*Vedi Tabella *)
				MB_BitStato[208]:=ModBus.MB_MASTER.ReceiveBuffer.Data[5].0; (*Vedi Tabella *)
				MB_BitStato[209]:=ModBus.MB_MASTER.ReceiveBuffer.Data[5].1; (*Vedi Tabella *)
				MB_BitStato[210]:=ModBus.MB_MASTER.ReceiveBuffer.Data[5].2; (*Vedi Tabella *)
				MB_BitStato[211]:=ModBus.MB_MASTER.ReceiveBuffer.Data[5].3; (*Vedi Tabella *)
				MB_BitStato[212]:=ModBus.MB_MASTER.ReceiveBuffer.Data[5].4; (*Vedi Tabella *)
				MB_BitStato[213]:=ModBus.MB_MASTER.ReceiveBuffer.Data[5].5; (*Vedi Tabella *)
				MB_BitStato[214]:=ModBus.MB_MASTER.ReceiveBuffer.Data[5].6; (*Vedi Tabella *)
				MB_BitStato[215]:=ModBus.MB_MASTER.ReceiveBuffer.Data[5].7; (*Vedi Tabella *)
				MB_BitStato[216]:=ModBus.MB_MASTER.ReceiveBuffer.Data[6].0; (*Vedi Tabella *)
				MB_BitStato[217]:=ModBus.MB_MASTER.ReceiveBuffer.Data[6].1; (*Vedi Tabella *)
				MB_BitStato[218]:=ModBus.MB_MASTER.ReceiveBuffer.Data[6].2; (*Vedi Tabella *)
				MB_BitStato[219]:=ModBus.MB_MASTER.ReceiveBuffer.Data[6].3; (*Vedi Tabella *)
				MB_BitStato[220]:=ModBus.MB_MASTER.ReceiveBuffer.Data[6].4; (*Vedi Tabella *)
				MB_BitStato[221]:=ModBus.MB_MASTER.ReceiveBuffer.Data[6].5; (*Vedi Tabella *)
				MB_BitStato[222]:=ModBus.MB_MASTER.ReceiveBuffer.Data[6].6; (*Vedi Tabella *)
				MB_BitStato[223]:=ModBus.MB_MASTER.ReceiveBuffer.Data[6].7; (*Vedi Tabella *)
				MB_BitStato[224]:=ModBus.MB_MASTER.ReceiveBuffer.Data[7].0; (*Vedi Tabella *)
				MB_BitStato[225]:=ModBus.MB_MASTER.ReceiveBuffer.Data[7].1; (*Vedi Tabella *)
				MB_BitStato[226]:=ModBus.MB_MASTER.ReceiveBuffer.Data[7].2; (*Vedi Tabella *)
				MB_BitStato[227]:=ModBus.MB_MASTER.ReceiveBuffer.Data[7].3; (*Vedi Tabella *)
				MB_BitStato[228]:=ModBus.MB_MASTER.ReceiveBuffer.Data[7].4; (*Vedi Tabella *)
				MB_BitStato[229]:=ModBus.MB_MASTER.ReceiveBuffer.Data[7].5; (*Vedi Tabella *)
				MB_BitStato[230]:=ModBus.MB_MASTER.ReceiveBuffer.Data[7].6; (*Vedi Tabella *)
				MB_BitStato[231]:=ModBus.MB_MASTER.ReceiveBuffer.Data[7].7; (*Vedi Tabella *)
				MB_BitStato[232]:=ModBus.MB_MASTER.ReceiveBuffer.Data[8].0; (*Vedi Tabella *)
				MB_BitStato[233]:=ModBus.MB_MASTER.ReceiveBuffer.Data[8].1; (*Vedi Tabella *)
				MB_BitStato[234]:=ModBus.MB_MASTER.ReceiveBuffer.Data[8].2; (*Vedi Tabella *)
				MB_BitStato[235]:=ModBus.MB_MASTER.ReceiveBuffer.Data[8].3; (*Vedi Tabella *)
				MB_BitStato[236]:=ModBus.MB_MASTER.ReceiveBuffer.Data[8].4; (*Vedi Tabella *)
				MB_BitStato[237]:=ModBus.MB_MASTER.ReceiveBuffer.Data[8].5; (*Vedi Tabella *)
				MB_BitStato[238]:=ModBus.MB_MASTER.ReceiveBuffer.Data[8].6; (*Vedi Tabella *)
				MB_BitStato[239]:=ModBus.MB_MASTER.ReceiveBuffer.Data[8].7; (*Vedi Tabella *)
				MB_BitStato[240]:=ModBus.MB_MASTER.ReceiveBuffer.Data[9].0; (*Vedi Tabella *)
				MB_BitStato[241]:=ModBus.MB_MASTER.ReceiveBuffer.Data[9].1; (*Vedi Tabella *)
				MB_BitStato[242]:=ModBus.MB_MASTER.ReceiveBuffer.Data[9].2; (*Vedi Tabella *)
				MB_BitStato[243]:=ModBus.MB_MASTER.ReceiveBuffer.Data[9].3; (*Vedi Tabella *)
				MB_BitStato[244]:=ModBus.MB_MASTER.ReceiveBuffer.Data[9].4; (*Vedi Tabella *)
				MB_BitStato[245]:=ModBus.MB_MASTER.ReceiveBuffer.Data[9].5; (*Vedi Tabella *)
				MB_BitStato[246]:=ModBus.MB_MASTER.ReceiveBuffer.Data[9].6; (*Vedi Tabella *)
				MB_BitStato[247]:=ModBus.MB_MASTER.ReceiveBuffer.Data[9].7; (*Vedi Tabella *)
				MB_BitStato[248]:=ModBus.MB_MASTER.ReceiveBuffer.Data[10].0; (*Vedi Tabella *)
				MB_BitStato[249]:=ModBus.MB_MASTER.ReceiveBuffer.Data[10].1; (*Vedi Tabella *)
				MB_BitStato[250]:=ModBus.MB_MASTER.ReceiveBuffer.Data[10].2; (*Vedi Tabella *)
				MB_BitStato[251]:=ModBus.MB_MASTER.ReceiveBuffer.Data[10].3; (*Vedi Tabella *)
				MB_BitStato[252]:=ModBus.MB_MASTER.ReceiveBuffer.Data[10].4; (*Vedi Tabella *)
				MB_BitStato[253]:=ModBus.MB_MASTER.ReceiveBuffer.Data[10].5; (*Vedi Tabella *)
				MB_BitStato[254]:=ModBus.MB_MASTER.ReceiveBuffer.Data[10].6; (*Vedi Tabella *)
				MB_BitStato[255]:=ModBus.MB_MASTER.ReceiveBuffer.Data[10].7; (*Vedi Tabella *)

				state:=140;

			END_IF
		END_IF

	140: (* Rispota Altri paramenti COIL *)
		IF NOT ModBus.MB_Start  THEN

			IF ModBus.MB_MASTER.MB_Error<>0 THEN
				state := 300;
			ELSE
				Modbus.MB_Query.SlaveAddress := Address;
				Modbus.MB_Query.FunctionCode := 2;
				ModBus.MB_Query.Read_StartAddress := 256;	(* richiedo lettura altri Parametri *)
				ModBus.MB_Query.Read_Quantity := 64;
				ModBus.MB_Start := TRUE;

				state:=145;
			END_IF
		END_IF
	145: (* Rispota Altri paramenti *)

		IF NOT ModBus.MB_Start  THEN

			IF ModBus.MB_MASTER.MB_Error<>0 THEN
				state := 300;
			ELSE

				MB_BitStato[256]:=ModBus.MB_MASTER.ReceiveBuffer.Data[3].0; (*Vedi Tabella *)
				MB_BitStato[257]:=ModBus.MB_MASTER.ReceiveBuffer.Data[3].1; (*Vedi Tabella *)
				MB_BitStato[258]:=ModBus.MB_MASTER.ReceiveBuffer.Data[3].2; (*Vedi Tabella *)
				MB_BitStato[259]:=ModBus.MB_MASTER.ReceiveBuffer.Data[3].3; (*Vedi Tabella *)
				MB_BitStato[260]:=ModBus.MB_MASTER.ReceiveBuffer.Data[3].4; (*Vedi Tabella *)
				MB_BitStato[261]:=ModBus.MB_MASTER.ReceiveBuffer.Data[3].5; (*Vedi Tabella *)
				MB_BitStato[262]:=ModBus.MB_MASTER.ReceiveBuffer.Data[3].6; (*Vedi Tabella *)
				MB_BitStato[263]:=ModBus.MB_MASTER.ReceiveBuffer.Data[3].7; (*Vedi Tabella *)
				MB_BitStato[264]:=ModBus.MB_MASTER.ReceiveBuffer.Data[4].0; (*Vedi Tabella *)
				MB_BitStato[265]:=ModBus.MB_MASTER.ReceiveBuffer.Data[4].1; (*Vedi Tabella *)
				MB_BitStato[266]:=ModBus.MB_MASTER.ReceiveBuffer.Data[4].2; (*Vedi Tabella *)
				MB_BitStato[267]:=ModBus.MB_MASTER.ReceiveBuffer.Data[4].3; (*Vedi Tabella *)
				MB_BitStato[268]:=ModBus.MB_MASTER.ReceiveBuffer.Data[4].4; (*Vedi Tabella *)
				MB_BitStato[269]:=ModBus.MB_MASTER.ReceiveBuffer.Data[4].5; (*Vedi Tabella *)
				MB_BitStato[270]:=ModBus.MB_MASTER.ReceiveBuffer.Data[4].6; (*Vedi Tabella *)
				MB_BitStato[271]:=ModBus.MB_MASTER.ReceiveBuffer.Data[4].7; (*Vedi Tabella *)
				MB_BitStato[272]:=ModBus.MB_MASTER.ReceiveBuffer.Data[5].0; (*Vedi Tabella *)
				MB_BitStato[273]:=ModBus.MB_MASTER.ReceiveBuffer.Data[5].1; (*Vedi Tabella *)
				MB_BitStato[274]:=ModBus.MB_MASTER.ReceiveBuffer.Data[5].2; (*Vedi Tabella *)
				MB_BitStato[275]:=ModBus.MB_MASTER.ReceiveBuffer.Data[5].3; (*Vedi Tabella *)
				MB_BitStato[276]:=ModBus.MB_MASTER.ReceiveBuffer.Data[5].4; (*Vedi Tabella *)
				MB_BitStato[277]:=ModBus.MB_MASTER.ReceiveBuffer.Data[5].5; (*Vedi Tabella *)
				MB_BitStato[278]:=ModBus.MB_MASTER.ReceiveBuffer.Data[5].6; (*Vedi Tabella *)
				MB_BitStato[279]:=ModBus.MB_MASTER.ReceiveBuffer.Data[5].7; (*Vedi Tabella *)
				MB_BitStato[280]:=ModBus.MB_MASTER.ReceiveBuffer.Data[6].0; (*Vedi Tabella *)
				MB_BitStato[281]:=ModBus.MB_MASTER.ReceiveBuffer.Data[6].1; (*Vedi Tabella *)
				MB_BitStato[282]:=ModBus.MB_MASTER.ReceiveBuffer.Data[6].2; (*Vedi Tabella *)
				MB_BitStato[283]:=ModBus.MB_MASTER.ReceiveBuffer.Data[6].3; (*Vedi Tabella *)
				MB_BitStato[284]:=ModBus.MB_MASTER.ReceiveBuffer.Data[6].4; (*Vedi Tabella *)
				MB_BitStato[285]:=ModBus.MB_MASTER.ReceiveBuffer.Data[6].5; (*Vedi Tabella *)
				MB_BitStato[286]:=ModBus.MB_MASTER.ReceiveBuffer.Data[6].6; (*Vedi Tabella *)
				MB_BitStato[287]:=ModBus.MB_MASTER.ReceiveBuffer.Data[6].7; (*Vedi Tabella *)
				MB_BitStato[288]:=ModBus.MB_MASTER.ReceiveBuffer.Data[7].0; (*Vedi Tabella *)
				MB_BitStato[289]:=ModBus.MB_MASTER.ReceiveBuffer.Data[7].1; (*Vedi Tabella *)
				MB_BitStato[290]:=ModBus.MB_MASTER.ReceiveBuffer.Data[7].2; (*Vedi Tabella *)
				MB_BitStato[291]:=ModBus.MB_MASTER.ReceiveBuffer.Data[7].3; (*Vedi Tabella *)
				MB_BitStato[292]:=ModBus.MB_MASTER.ReceiveBuffer.Data[7].4; (*Vedi Tabella *)
				MB_BitStato[293]:=ModBus.MB_MASTER.ReceiveBuffer.Data[7].5; (*Vedi Tabella *)
				MB_BitStato[294]:=ModBus.MB_MASTER.ReceiveBuffer.Data[7].6; (*Vedi Tabella *)
				MB_BitStato[295]:=ModBus.MB_MASTER.ReceiveBuffer.Data[7].7; (*Vedi Tabella *)
				MB_BitStato[296]:=ModBus.MB_MASTER.ReceiveBuffer.Data[8].0; (*Vedi Tabella *)
				MB_BitStato[297]:=ModBus.MB_MASTER.ReceiveBuffer.Data[8].1; (*Vedi Tabella *)
				MB_BitStato[298]:=ModBus.MB_MASTER.ReceiveBuffer.Data[8].2; (*Vedi Tabella *)
				MB_BitStato[299]:=ModBus.MB_MASTER.ReceiveBuffer.Data[8].3; (*Vedi Tabella *)
				MB_BitStato[300]:=ModBus.MB_MASTER.ReceiveBuffer.Data[8].4; (*Vedi Tabella *)
				MB_BitStato[301]:=ModBus.MB_MASTER.ReceiveBuffer.Data[8].5; (*Vedi Tabella *)
				MB_BitStato[302]:=ModBus.MB_MASTER.ReceiveBuffer.Data[8].6; (*Vedi Tabella *)
				MB_BitStato[303]:=ModBus.MB_MASTER.ReceiveBuffer.Data[8].7; (*Vedi Tabella *)
				MB_BitStato[304]:=ModBus.MB_MASTER.ReceiveBuffer.Data[9].0; (*Vedi Tabella *)
				MB_BitStato[305]:=ModBus.MB_MASTER.ReceiveBuffer.Data[9].1; (*Vedi Tabella *)
				MB_BitStato[306]:=ModBus.MB_MASTER.ReceiveBuffer.Data[9].2; (*Vedi Tabella *)
				MB_BitStato[307]:=ModBus.MB_MASTER.ReceiveBuffer.Data[9].3; (*Vedi Tabella *)
				MB_BitStato[308]:=ModBus.MB_MASTER.ReceiveBuffer.Data[9].4; (*Vedi Tabella *)
				MB_BitStato[309]:=ModBus.MB_MASTER.ReceiveBuffer.Data[9].5; (*Vedi Tabella *)
				MB_BitStato[310]:=ModBus.MB_MASTER.ReceiveBuffer.Data[9].6; (*Vedi Tabella *)
				MB_BitStato[311]:=ModBus.MB_MASTER.ReceiveBuffer.Data[9].7; (*Vedi Tabella *)
				MB_BitStato[312]:=ModBus.MB_MASTER.ReceiveBuffer.Data[10].0; (*Vedi Tabella *)
				MB_BitStato[313]:=ModBus.MB_MASTER.ReceiveBuffer.Data[10].1; (*Vedi Tabella *)
				MB_BitStato[314]:=ModBus.MB_MASTER.ReceiveBuffer.Data[10].2; (*Vedi Tabella *)
				MB_BitStato[315]:=ModBus.MB_MASTER.ReceiveBuffer.Data[10].3; (*Vedi Tabella *)
				MB_BitStato[316]:=ModBus.MB_MASTER.ReceiveBuffer.Data[10].4; (*Vedi Tabella *)
				MB_BitStato[317]:=ModBus.MB_MASTER.ReceiveBuffer.Data[10].5; (*Vedi Tabella *)
				MB_BitStato[318]:=ModBus.MB_MASTER.ReceiveBuffer.Data[10].6; (*Vedi Tabella *)
				MB_BitStato[319]:=ModBus.MB_MASTER.ReceiveBuffer.Data[10].7; (*Vedi Tabella *)

				state:=160;

			END_IF
		END_IF

	160: (* Rispota Altri paramenti COIL *)
		IF NOT ModBus.MB_Start  THEN

			IF ModBus.MB_MASTER.MB_Error<>0 THEN
				state := 300;
			ELSE
				Modbus.MB_Query.SlaveAddress := Address;
				Modbus.MB_Query.FunctionCode := 2;
				ModBus.MB_Query.Read_StartAddress := 320;	(* richiedo lettura altri Parametri *)
				ModBus.MB_Query.Read_Quantity := 64;
				ModBus.MB_Start := TRUE;

				state:=165;
			END_IF
		END_IF
	165: (* Rispota Altri paramenti *)

		IF NOT ModBus.MB_Start  THEN

			IF ModBus.MB_MASTER.MB_Error<>0 THEN
				state := 300;
			ELSE

				MB_BitStato[320]:=ModBus.MB_MASTER.ReceiveBuffer.Data[3].0; (*Vedi Tabella *)
				MB_BitStato[321]:=ModBus.MB_MASTER.ReceiveBuffer.Data[3].1; (*Vedi Tabella *)
				MB_BitStato[322]:=ModBus.MB_MASTER.ReceiveBuffer.Data[3].2; (*Vedi Tabella *)
				MB_BitStato[323]:=ModBus.MB_MASTER.ReceiveBuffer.Data[3].3; (*Vedi Tabella *)
				MB_BitStato[324]:=ModBus.MB_MASTER.ReceiveBuffer.Data[3].4; (*Vedi Tabella *)
				MB_BitStato[325]:=ModBus.MB_MASTER.ReceiveBuffer.Data[3].5; (*Vedi Tabella *)
				MB_BitStato[326]:=ModBus.MB_MASTER.ReceiveBuffer.Data[3].6; (*Vedi Tabella *)
				MB_BitStato[327]:=ModBus.MB_MASTER.ReceiveBuffer.Data[3].7; (*Vedi Tabella *)
				MB_BitStato[328]:=ModBus.MB_MASTER.ReceiveBuffer.Data[4].0; (*Vedi Tabella *)
				MB_BitStato[329]:=ModBus.MB_MASTER.ReceiveBuffer.Data[4].1; (*Vedi Tabella *)
				MB_BitStato[330]:=ModBus.MB_MASTER.ReceiveBuffer.Data[4].2; (*Vedi Tabella *)
				MB_BitStato[331]:=ModBus.MB_MASTER.ReceiveBuffer.Data[4].3; (*Vedi Tabella *)
				MB_BitStato[332]:=ModBus.MB_MASTER.ReceiveBuffer.Data[4].4; (*Vedi Tabella *)
				MB_BitStato[333]:=ModBus.MB_MASTER.ReceiveBuffer.Data[4].5; (*Vedi Tabella *)
				MB_BitStato[334]:=ModBus.MB_MASTER.ReceiveBuffer.Data[4].6; (*Vedi Tabella *)
				MB_BitStato[335]:=ModBus.MB_MASTER.ReceiveBuffer.Data[4].7; (*Vedi Tabella *)
				MB_BitStato[336]:=ModBus.MB_MASTER.ReceiveBuffer.Data[5].0; (*Vedi Tabella *)
				MB_BitStato[337]:=ModBus.MB_MASTER.ReceiveBuffer.Data[5].1; (*Vedi Tabella *)
				MB_BitStato[338]:=ModBus.MB_MASTER.ReceiveBuffer.Data[5].2; (*Vedi Tabella *)
				MB_BitStato[339]:=ModBus.MB_MASTER.ReceiveBuffer.Data[5].3; (*Vedi Tabella *)
				MB_BitStato[340]:=ModBus.MB_MASTER.ReceiveBuffer.Data[5].4; (*Vedi Tabella *)
				MB_BitStato[341]:=ModBus.MB_MASTER.ReceiveBuffer.Data[5].5; (*Vedi Tabella *)
				MB_BitStato[342]:=ModBus.MB_MASTER.ReceiveBuffer.Data[5].6; (*Vedi Tabella *)
				MB_BitStato[343]:=ModBus.MB_MASTER.ReceiveBuffer.Data[5].7; (*Vedi Tabella *)
				MB_BitStato[344]:=ModBus.MB_MASTER.ReceiveBuffer.Data[6].0; (*Vedi Tabella *)
				MB_BitStato[345]:=ModBus.MB_MASTER.ReceiveBuffer.Data[6].1; (*Vedi Tabella *)
				MB_BitStato[346]:=ModBus.MB_MASTER.ReceiveBuffer.Data[6].2; (*Vedi Tabella *)
				MB_BitStato[347]:=ModBus.MB_MASTER.ReceiveBuffer.Data[6].3; (*Vedi Tabella *)
				MB_BitStato[348]:=ModBus.MB_MASTER.ReceiveBuffer.Data[6].4; (*Vedi Tabella *)
				MB_BitStato[349]:=ModBus.MB_MASTER.ReceiveBuffer.Data[6].5; (*Vedi Tabella *)
				MB_BitStato[350]:=ModBus.MB_MASTER.ReceiveBuffer.Data[6].6; (*Vedi Tabella *)
				MB_BitStato[351]:=ModBus.MB_MASTER.ReceiveBuffer.Data[6].7; (*Vedi Tabella *)
				MB_BitStato[352]:=ModBus.MB_MASTER.ReceiveBuffer.Data[7].0; (*Vedi Tabella *)
				MB_BitStato[353]:=ModBus.MB_MASTER.ReceiveBuffer.Data[7].1; (*Vedi Tabella *)
				MB_BitStato[354]:=ModBus.MB_MASTER.ReceiveBuffer.Data[7].2; (*Vedi Tabella *)
				MB_BitStato[355]:=ModBus.MB_MASTER.ReceiveBuffer.Data[7].3; (*Vedi Tabella *)
				MB_BitStato[356]:=ModBus.MB_MASTER.ReceiveBuffer.Data[7].4; (*Vedi Tabella *)
				MB_BitStato[357]:=ModBus.MB_MASTER.ReceiveBuffer.Data[7].5; (*Vedi Tabella *)
	(*			MB_BitStato[359]:=ModBus.MB_MASTER.ReceiveBuffer.Data[7].6; (*Vedi Tabella *)
				MB_BitStato[360]:=ModBus.MB_MASTER.ReceiveBuffer.Data[7].7; (*Vedi Tabella *)
				MB_BitStato[40]:=ModBus.MB_MASTER.ReceiveBuffer.Data[8].0; (*Vedi Tabella *)
				MB_BitStato[41]:=ModBus.MB_MASTER.ReceiveBuffer.Data[8].1; (*Vedi Tabella *)
				MB_BitStato[42]:=ModBus.MB_MASTER.ReceiveBuffer.Data[8].2; (*Vedi Tabella *)
				MB_BitStato[43]:=ModBus.MB_MASTER.ReceiveBuffer.Data[8].3; (*Vedi Tabella *)
				MB_BitStato[44]:=ModBus.MB_MASTER.ReceiveBuffer.Data[8].4; (*Vedi Tabella *)
				MB_BitStato[45]:=ModBus.MB_MASTER.ReceiveBuffer.Data[8].5; (*Vedi Tabella *)
				MB_BitStato[46]:=ModBus.MB_MASTER.ReceiveBuffer.Data[8].6; (*Vedi Tabella *)
				MB_BitStato[47]:=ModBus.MB_MASTER.ReceiveBuffer.Data[8].7; (*Vedi Tabella *)
				MB_BitStato[48]:=ModBus.MB_MASTER.ReceiveBuffer.Data[9].0; (*Vedi Tabella *)
				MB_BitStato[49]:=ModBus.MB_MASTER.ReceiveBuffer.Data[9].1; (*Vedi Tabella *)
				MB_BitStato[50]:=ModBus.MB_MASTER.ReceiveBuffer.Data[9].2; (*Vedi Tabella *)
				MB_BitStato[51]:=ModBus.MB_MASTER.ReceiveBuffer.Data[9].3; (*Vedi Tabella *)
				MB_BitStato[52]:=ModBus.MB_MASTER.ReceiveBuffer.Data[9].4; (*Vedi Tabella *)
				MB_BitStato[53]:=ModBus.MB_MASTER.ReceiveBuffer.Data[9].5; (*Vedi Tabella *)
				MB_BitStato[54]:=ModBus.MB_MASTER.ReceiveBuffer.Data[9].6; (*Vedi Tabella *)
				MB_BitStato[55]:=ModBus.MB_MASTER.ReceiveBuffer.Data[9].7; (*Vedi Tabella *)
				MB_BitStato[56]:=ModBus.MB_MASTER.ReceiveBuffer.Data[10].0; (*Vedi Tabella *)
				MB_BitStato[57]:=ModBus.MB_MASTER.ReceiveBuffer.Data[10].1; (*Vedi Tabella *)
				MB_BitStato[58]:=ModBus.MB_MASTER.ReceiveBuffer.Data[10].2; (*Vedi Tabella *)
				MB_BitStato[59]:=ModBus.MB_MASTER.ReceiveBuffer.Data[10].3; (*Vedi Tabella *)
				MB_BitStato[60]:=ModBus.MB_MASTER.ReceiveBuffer.Data[10].4; (*Vedi Tabella *)
				MB_BitStato[61]:=ModBus.MB_MASTER.ReceiveBuffer.Data[10].5; (*Vedi Tabella *)
				MB_BitStato[62]:=ModBus.MB_MASTER.ReceiveBuffer.Data[10].6; (*Vedi Tabella *)
				MB_BitStato[63]:=ModBus.MB_MASTER.ReceiveBuffer.Data[10].7; (*Vedi Tabella *)
*)
				state:=170;

			END_IF
		END_IF





	170: (* Rispota Altri paramenti COIL *)
		IF NOT ModBus.MB_Start  THEN

			IF ModBus.MB_MASTER.MB_Error<>0 THEN
				state := 300;
			ELSE
				Modbus.MB_Query.SlaveAddress := Address;
				Modbus.MB_Query.FunctionCode := 1;
				ModBus.MB_Query.Read_StartAddress := 0;	(* richiedo lettura altri Parametri *)
				ModBus.MB_Query.Read_Quantity := 64;
				ModBus.MB_Start := TRUE;

				state:=171;
			END_IF
		END_IF
	171: (* Rispota Altri paramenti *)

		IF NOT ModBus.MB_Start  THEN

			IF ModBus.MB_MASTER.MB_Error<>0 THEN
				state := 300;
			ELSE

				MB_BitStatoCoil[0]:=ModBus.MB_MASTER.ReceiveBuffer.Data[3].0; (*Vedi Tabella *)
				MB_BitStatoCoil[1]:=ModBus.MB_MASTER.ReceiveBuffer.Data[3].1; (*Vedi Tabella *)
				MB_BitStatoCoil[2]:=ModBus.MB_MASTER.ReceiveBuffer.Data[3].2; (*Vedi Tabella *)
				MB_BitStatoCoil[3]:=ModBus.MB_MASTER.ReceiveBuffer.Data[3].3; (*Vedi Tabella *)
				MB_BitStatoCoil[4]:=ModBus.MB_MASTER.ReceiveBuffer.Data[3].4; (*Vedi Tabella *)
				MB_BitStatoCoil[5]:=ModBus.MB_MASTER.ReceiveBuffer.Data[3].5; (*Vedi Tabella *)
				MB_BitStatoCoil[6]:=ModBus.MB_MASTER.ReceiveBuffer.Data[3].6; (*Vedi Tabella *)
				MB_BitStatoCoil[7]:=ModBus.MB_MASTER.ReceiveBuffer.Data[3].7; (*Vedi Tabella *)
				MB_BitStatoCoil[8]:=ModBus.MB_MASTER.ReceiveBuffer.Data[4].0; (*Vedi Tabella *)
				MB_BitStatoCoil[9]:=ModBus.MB_MASTER.ReceiveBuffer.Data[4].1; (*Vedi Tabella *)
				MB_BitStatoCoil[10]:=ModBus.MB_MASTER.ReceiveBuffer.Data[4].2; (*Vedi Tabella *)
				MB_BitStatoCoil[11]:=ModBus.MB_MASTER.ReceiveBuffer.Data[4].3; (*Vedi Tabella *)
				MB_BitStatoCoil[12]:=ModBus.MB_MASTER.ReceiveBuffer.Data[4].4; (*Vedi Tabella *)
				MB_BitStatoCoil[13]:=ModBus.MB_MASTER.ReceiveBuffer.Data[4].5; (*Vedi Tabella *)
				MB_BitStatoCoil[14]:=ModBus.MB_MASTER.ReceiveBuffer.Data[4].6; (*Vedi Tabella *)
				MB_BitStatoCoil[15]:=ModBus.MB_MASTER.ReceiveBuffer.Data[4].7; (*Vedi Tabella *)
				MB_BitStatoCoil[16]:=ModBus.MB_MASTER.ReceiveBuffer.Data[5].0; (*Vedi Tabella *)
				MB_BitStatoCoil[17]:=ModBus.MB_MASTER.ReceiveBuffer.Data[5].1; (*Vedi Tabella *)
				MB_BitStatoCoil[18]:=ModBus.MB_MASTER.ReceiveBuffer.Data[5].2; (*Vedi Tabella *)
				MB_BitStatoCoil[19]:=ModBus.MB_MASTER.ReceiveBuffer.Data[5].3; (*Vedi Tabella *)
				MB_BitStatoCoil[20]:=ModBus.MB_MASTER.ReceiveBuffer.Data[5].4; (*Vedi Tabella *)
				MB_BitStatoCoil[21]:=ModBus.MB_MASTER.ReceiveBuffer.Data[5].5; (*Vedi Tabella *)
				MB_BitStatoCoil[22]:=ModBus.MB_MASTER.ReceiveBuffer.Data[5].6; (*Vedi Tabella *)
				MB_BitStatoCoil[23]:=ModBus.MB_MASTER.ReceiveBuffer.Data[5].7; (*Vedi Tabella *)
				MB_BitStatoCoil[24]:=ModBus.MB_MASTER.ReceiveBuffer.Data[6].0; (*Vedi Tabella *)
				MB_BitStatoCoil[25]:=ModBus.MB_MASTER.ReceiveBuffer.Data[6].1; (*Vedi Tabella *)
				MB_BitStatoCoil[26]:=ModBus.MB_MASTER.ReceiveBuffer.Data[6].2; (*Vedi Tabella *)
				MB_BitStatoCoil[27]:=ModBus.MB_MASTER.ReceiveBuffer.Data[6].3; (*Vedi Tabella *)
				MB_BitStatoCoil[28]:=ModBus.MB_MASTER.ReceiveBuffer.Data[6].4; (*Vedi Tabella *)
				MB_BitStatoCoil[29]:=ModBus.MB_MASTER.ReceiveBuffer.Data[6].5; (*Vedi Tabella *)
				MB_BitStatoCoil[30]:=ModBus.MB_MASTER.ReceiveBuffer.Data[6].6; (*Vedi Tabella *)
				MB_BitStatoCoil[31]:=ModBus.MB_MASTER.ReceiveBuffer.Data[6].7; (*Vedi Tabella *)
				MB_BitStatoCoil[32]:=ModBus.MB_MASTER.ReceiveBuffer.Data[7].0; (*Vedi Tabella *)
				MB_BitStatoCoil[33]:=ModBus.MB_MASTER.ReceiveBuffer.Data[7].1; (*Vedi Tabella *)
				MB_BitStatoCoil[34]:=ModBus.MB_MASTER.ReceiveBuffer.Data[7].2; (*Vedi Tabella *)
				MB_BitStatoCoil[35]:=ModBus.MB_MASTER.ReceiveBuffer.Data[7].3; (*Vedi Tabella *)
				MB_BitStatoCoil[36]:=ModBus.MB_MASTER.ReceiveBuffer.Data[7].4; (*Vedi Tabella *)
				MB_BitStatoCoil[37]:=ModBus.MB_MASTER.ReceiveBuffer.Data[7].5; (*Vedi Tabella *)
				MB_BitStatoCoil[38]:=ModBus.MB_MASTER.ReceiveBuffer.Data[7].6; (*Vedi Tabella *)
				MB_BitStatoCoil[39]:=ModBus.MB_MASTER.ReceiveBuffer.Data[7].7; (*Vedi Tabella *)
				MB_BitStatoCoil[40]:=ModBus.MB_MASTER.ReceiveBuffer.Data[8].0; (*Vedi Tabella *)
				MB_BitStatoCoil[41]:=ModBus.MB_MASTER.ReceiveBuffer.Data[8].1; (*Vedi Tabella *)
				MB_BitStatoCoil[42]:=ModBus.MB_MASTER.ReceiveBuffer.Data[8].2; (*Vedi Tabella *)
				MB_BitStatoCoil[43]:=ModBus.MB_MASTER.ReceiveBuffer.Data[8].3; (*Vedi Tabella *)
				MB_BitStatoCoil[44]:=ModBus.MB_MASTER.ReceiveBuffer.Data[8].4; (*Vedi Tabella *)
				MB_BitStatoCoil[45]:=ModBus.MB_MASTER.ReceiveBuffer.Data[8].5; (*Vedi Tabella *)
				MB_BitStatoCoil[46]:=ModBus.MB_MASTER.ReceiveBuffer.Data[8].6; (*Vedi Tabella *)
				MB_BitStatoCoil[47]:=ModBus.MB_MASTER.ReceiveBuffer.Data[8].7; (*Vedi Tabella *)
				MB_BitStatoCoil[48]:=ModBus.MB_MASTER.ReceiveBuffer.Data[9].0; (*Vedi Tabella *)
				MB_BitStatoCoil[49]:=ModBus.MB_MASTER.ReceiveBuffer.Data[9].1; (*Vedi Tabella *)
				MB_BitStatoCoil[50]:=ModBus.MB_MASTER.ReceiveBuffer.Data[9].2; (*Vedi Tabella *)
				MB_BitStatoCoil[51]:=ModBus.MB_MASTER.ReceiveBuffer.Data[9].3; (*Vedi Tabella *)
				MB_BitStatoCoil[52]:=ModBus.MB_MASTER.ReceiveBuffer.Data[9].4; (*Vedi Tabella *)
				MB_BitStatoCoil[53]:=ModBus.MB_MASTER.ReceiveBuffer.Data[9].5; (*Vedi Tabella *)
				MB_BitStatoCoil[54]:=ModBus.MB_MASTER.ReceiveBuffer.Data[9].6; (*Vedi Tabella *)
				MB_BitStatoCoil[55]:=ModBus.MB_MASTER.ReceiveBuffer.Data[9].7; (*Vedi Tabella *)
				MB_BitStatoCoil[56]:=ModBus.MB_MASTER.ReceiveBuffer.Data[10].0; (*Vedi Tabella *)
				MB_BitStatoCoil[57]:=ModBus.MB_MASTER.ReceiveBuffer.Data[10].1; (*Vedi Tabella *)
				MB_BitStatoCoil[58]:=ModBus.MB_MASTER.ReceiveBuffer.Data[10].2; (*Vedi Tabella *)
				MB_BitStatoCoil[59]:=ModBus.MB_MASTER.ReceiveBuffer.Data[10].3; (*Vedi Tabella *)
				MB_BitStatoCoil[60]:=ModBus.MB_MASTER.ReceiveBuffer.Data[10].4; (*Vedi Tabella *)
				MB_BitStatoCoil[61]:=ModBus.MB_MASTER.ReceiveBuffer.Data[10].5; (*Vedi Tabella *)
				MB_BitStatoCoil[62]:=ModBus.MB_MASTER.ReceiveBuffer.Data[10].6; (*Vedi Tabella *)
				MB_BitStatoCoil[63]:=ModBus.MB_MASTER.ReceiveBuffer.Data[10].7; (*Vedi Tabella *)
				MB_BitStatoCoil[64]:=ModBus.MB_MASTER.ReceiveBuffer.Data[11].0; (*Vedi Tabella *)
				MB_BitStatoCoil[65]:=ModBus.MB_MASTER.ReceiveBuffer.Data[11].1; (*Vedi Tabella *)
				MB_BitStatoCoil[66]:=ModBus.MB_MASTER.ReceiveBuffer.Data[1].2; (*Vedi Tabella *)
				MB_BitStatoCoil[67]:=ModBus.MB_MASTER.ReceiveBuffer.Data[11].3; (*Vedi Tabella *)
				MB_BitStatoCoil[68]:=ModBus.MB_MASTER.ReceiveBuffer.Data[11].4; (*Vedi Tabella *)
				MB_BitStatoCoil[69]:=ModBus.MB_MASTER.ReceiveBuffer.Data[11].5; (*Vedi Tabella *)
				MB_BitStatoCoil[70]:=ModBus.MB_MASTER.ReceiveBuffer.Data[11].6; (*Vedi Tabella *)
				MB_BitStatoCoil[71]:=ModBus.MB_MASTER.ReceiveBuffer.Data[11].7; (*Vedi Tabella *)
				state:=290 ;   (*********************************************************************************)

			END_IF
		END_IF


		200:    (* Scrittura BOOL Abilita UTA 01 *)
		IF NOT ModBus.MB_Start THEN
			IF ModBus.MB_MASTER.MB_Error<>0 THEN (*OR ModBus.MB_MASTER.MB_Error<>0 THEN*)
				state := 300;
			ELSE
				AddressDaScrivere:=19;
				IF ScriviRUN_UTA01 THEN
					Modbus.MB_Query.FunctionCode := 5;
					Modbus.MB_Query.SlaveAddress := Address;
					ModBus.MB_Query.Write_StartAddress := AddressDaScrivere;
					ModBus.MB_Query.Write_Quantity :=1;
					ModBus.MB_Query.Write_Data[0] := BOOL_TO_WORD(Abilita_UTA01);
					ModBus.MB_Start := TRUE;
					IF 	MB_BitStatoCoil[AddressDaScrivere]=(Abilita_UTA01) THEN
						ScriviRUN_UTA01:=FALSE;
					END_IF
					state := 201;
				ELSE
					state := 201;
				END_IF
			END_IF
		END_IF

		201:    (* Scrittura BOOL Abilita UTA 02 *)
		IF NOT ModBus.MB_Start THEN
			IF ModBus.MB_MASTER.MB_Error<>0 THEN (*OR ModBus.MB_MASTER.MB_Error<>0 THEN*)
				state := 300;
			ELSE
				AddressDaScrivere:=20;
				IF ScriviRUN_UTA02 THEN
					Modbus.MB_Query.FunctionCode := 5;
					Modbus.MB_Query.SlaveAddress := Address;
					ModBus.MB_Query.Write_StartAddress := AddressDaScrivere;
					ModBus.MB_Query.Write_Quantity :=1;
					ModBus.MB_Query.Write_Data[0] := BOOL_TO_WORD(Abilita_UTA02);
					ModBus.MB_Start := TRUE;
					IF 	MB_BitStatoCoil[AddressDaScrivere]=(Abilita_UTA02) THEN
						ScriviRUN_UTA02:=FALSE;
					END_IF
					state := 202;
				ELSE
					state := 202;
				END_IF
			END_IF
		END_IF

		202:    (* Scrittura BOOL Abilita UTA 03 *)
		IF NOT ModBus.MB_Start THEN
			IF ModBus.MB_MASTER.MB_Error<>0 THEN (*OR ModBus.MB_MASTER.MB_Error<>0 THEN*)
				state := 300;
			ELSE
				AddressDaScrivere:=21;
				IF ScriviRUN_UTA03 THEN
					Modbus.MB_Query.FunctionCode := 5;
					Modbus.MB_Query.SlaveAddress := Address;
					ModBus.MB_Query.Write_StartAddress := AddressDaScrivere;
					ModBus.MB_Query.Write_Quantity :=1;
					ModBus.MB_Query.Write_Data[0] := BOOL_TO_WORD(Abilita_UTA03);
					ModBus.MB_Start := TRUE;
					IF 	MB_BitStatoCoil[AddressDaScrivere]=(Abilita_UTA03) THEN
						ScriviRUN_UTA03:=FALSE;
					END_IF
					state := 203;
				ELSE
					state := 203;
				END_IF
			END_IF
		END_IF

		203:    (* Scrittura BOOL Abilita UTA 04 *)
		IF NOT ModBus.MB_Start THEN
			IF ModBus.MB_MASTER.MB_Error<>0 THEN (*OR ModBus.MB_MASTER.MB_Error<>0 THEN*)
				state := 300;
			ELSE
				AddressDaScrivere:=22;
				IF ScriviRUN_UTA04 THEN
					Modbus.MB_Query.FunctionCode := 5;
					Modbus.MB_Query.SlaveAddress := Address;
					ModBus.MB_Query.Write_StartAddress := AddressDaScrivere;
					ModBus.MB_Query.Write_Quantity :=1;
					ModBus.MB_Query.Write_Data[0] := BOOL_TO_WORD(Abilita_UTA04);
					ModBus.MB_Start := TRUE;
					IF 	MB_BitStatoCoil[AddressDaScrivere]=(Abilita_UTA04) THEN
						ScriviRUN_UTA04:=FALSE;
					END_IF
					state := 204;
				ELSE
					state := 204;
				END_IF
			END_IF
		END_IF

		204:    (* Scrittura BOOL Abilita UTA 05 *)
		IF NOT ModBus.MB_Start THEN
			IF ModBus.MB_MASTER.MB_Error<>0 THEN (*OR ModBus.MB_MASTER.MB_Error<>0 THEN*)
				state := 300;
			ELSE
				AddressDaScrivere:=23;
				IF ScriviRUN_UTA05 THEN
					Modbus.MB_Query.FunctionCode := 5;
					Modbus.MB_Query.SlaveAddress := Address;
					ModBus.MB_Query.Write_StartAddress := AddressDaScrivere;
					ModBus.MB_Query.Write_Quantity :=1;
					ModBus.MB_Query.Write_Data[0] := BOOL_TO_WORD(Abilita_UTA05);
					ModBus.MB_Start := TRUE;
					IF 	MB_BitStatoCoil[AddressDaScrivere]=(Abilita_UTA05) THEN
						ScriviRUN_UTA05:=FALSE;
					END_IF
					state := 205;
				ELSE
					state := 205;
				END_IF
			END_IF
		END_IF

		205:    (* Scrittura BOOL Abilita UTA 06 *)
		IF NOT ModBus.MB_Start THEN
			IF ModBus.MB_MASTER.MB_Error<>0 THEN (*OR ModBus.MB_MASTER.MB_Error<>0 THEN*)
				state := 300;
			ELSE
				AddressDaScrivere:=1;
				IF ScriviRUN_UTA06 THEN
					Modbus.MB_Query.FunctionCode := 5;
					Modbus.MB_Query.SlaveAddress := Address;
					ModBus.MB_Query.Write_StartAddress := AddressDaScrivere;
					ModBus.MB_Query.Write_Quantity :=1;
					ModBus.MB_Query.Write_Data[0] := BOOL_TO_WORD(Abilita_UTA06);
					ModBus.MB_Start := TRUE;
					IF 	MB_BitStatoCoil[AddressDaScrivere]=(Abilita_UTA06) THEN
						ScriviRUN_UTA06:=FALSE;
					END_IF
					state := 206;
				ELSE
					state := 206;
				END_IF
			END_IF
		END_IF

		206:    (* Scrittura BOOL Abilita UTA 07 *)
		IF NOT ModBus.MB_Start THEN
			IF ModBus.MB_MASTER.MB_Error<>0 THEN (*OR ModBus.MB_MASTER.MB_Error<>0 THEN*)
				state := 300;
			ELSE
				AddressDaScrivere:=2;
				IF ScriviRUN_UTA07 THEN
					Modbus.MB_Query.FunctionCode := 5;
					Modbus.MB_Query.SlaveAddress := Address;
					ModBus.MB_Query.Write_StartAddress := AddressDaScrivere;
					ModBus.MB_Query.Write_Quantity :=1;
					ModBus.MB_Query.Write_Data[0] := BOOL_TO_WORD(Abilita_UTA07);
					ModBus.MB_Start := TRUE;
					IF 	MB_BitStatoCoil[AddressDaScrivere]=(Abilita_UTA07) THEN
						ScriviRUN_UTA07:=FALSE;
					END_IF
					state := 207;
				ELSE
					state := 207;
				END_IF
			END_IF
		END_IF

		207:    (* Scrittura BOOL Abilita UTA 08 *)
		IF NOT ModBus.MB_Start THEN
			IF ModBus.MB_MASTER.MB_Error<>0 THEN (*OR ModBus.MB_MASTER.MB_Error<>0 THEN*)
				state := 300;
			ELSE
				AddressDaScrivere:=10;
				IF ScriviRUN_UTA08 THEN
					Modbus.MB_Query.FunctionCode := 5;
					Modbus.MB_Query.SlaveAddress := Address;
					ModBus.MB_Query.Write_StartAddress := AddressDaScrivere;
					ModBus.MB_Query.Write_Quantity :=1;
					ModBus.MB_Query.Write_Data[0] := BOOL_TO_WORD(Abilita_UTA08);
					ModBus.MB_Start := TRUE;
					IF 	MB_BitStatoCoil[AddressDaScrivere]=(Abilita_UTA08) THEN
						ScriviRUN_UTA08:=FALSE;
					END_IF
					state := 208;
				ELSE
					state := 208;
				END_IF
			END_IF
		END_IF

		208:    (* Scrittura BOOL Abilita UTA 09 *)
		IF NOT ModBus.MB_Start THEN
			IF ModBus.MB_MASTER.MB_Error<>0 THEN (*OR ModBus.MB_MASTER.MB_Error<>0 THEN*)
				state := 300;
			ELSE
				AddressDaScrivere:=11;
				IF ScriviRUN_UTA09 THEN
					Modbus.MB_Query.FunctionCode := 5;
					Modbus.MB_Query.SlaveAddress := Address;
					ModBus.MB_Query.Write_StartAddress := AddressDaScrivere;
					ModBus.MB_Query.Write_Quantity :=1;
					ModBus.MB_Query.Write_Data[0] := BOOL_TO_WORD(Abilita_UTA09);
					ModBus.MB_Start := TRUE;
					IF 	MB_BitStatoCoil[AddressDaScrivere]=(Abilita_UTA09) THEN
						ScriviRUN_UTA09:=FALSE;
					END_IF
					state := 209;
				ELSE
					state := 209;
				END_IF
			END_IF
		END_IF


		209:    (* Scrittura BOOL Abilita UTA 10 *)
		IF NOT ModBus.MB_Start THEN
			IF ModBus.MB_MASTER.MB_Error<>0 THEN (*OR ModBus.MB_MASTER.MB_Error<>0 THEN*)
				state := 300;
			ELSE
				AddressDaScrivere:=65;
				IF ScriviRUN_UTA10 THEN
					Modbus.MB_Query.FunctionCode := 5;
					Modbus.MB_Query.SlaveAddress := Address;
					ModBus.MB_Query.Write_StartAddress := AddressDaScrivere;
					ModBus.MB_Query.Write_Quantity :=1;
					ModBus.MB_Query.Write_Data[0] := BOOL_TO_WORD(Abilita_UTA10);
					ModBus.MB_Start := TRUE;
					IF 	MB_BitStatoCoil[AddressDaScrivere]=(Abilita_UTA10) THEN
						ScriviRUN_UTA10:=FALSE;
					END_IF
					state := 211;
				ELSE
					state := 211;
				END_IF
			END_IF
		END_IF

(*		210:    (* Scrittura BOOL Abilita UTA 11 *)
		IF NOT ModBus.MB_Start THEN
			IF ModBus.MB_MASTER.MB_Error<>0 THEN (*OR ModBus.MB_MASTER.MB_Error<>0 THEN*)
				state := 300;
			ELSE
				AddressDaScrivere:=65;
				IF ScriviRUN_UTA11 THEN
					Modbus.MB_Query.FunctionCode := 5;
					Modbus.MB_Query.SlaveAddress := Address;
					ModBus.MB_Query.Write_StartAddress := AddressDaScrivere;
					ModBus.MB_Query.Write_Quantity :=1;
					ModBus.MB_Query.Write_Data[0] := Abilita_UTA11;
					ModBus.MB_Start := TRUE;
					IF 	MB_BitStatoCoil[AddressDaScrivere]=WORD_TO_BOOL(Abilita_UTA11) THEN
						ScriviRUN_UTA11:=FALSE;
					END_IF
					state := 211;
				ELSE
					state := 211;
				END_IF
			END_IF
		END_IF
*)

		211:    (* Scrittura BOOL Abilita UTA 12 *)
		IF NOT ModBus.MB_Start THEN
			IF ModBus.MB_MASTER.MB_Error<>0 THEN (*OR ModBus.MB_MASTER.MB_Error<>0 THEN*)
				state := 300;
			ELSE
				AddressDaScrivere:=14;
				IF ScriviRUN_UTA12 THEN
					Modbus.MB_Query.FunctionCode := 5;
					Modbus.MB_Query.SlaveAddress := Address;
					ModBus.MB_Query.Write_StartAddress := AddressDaScrivere;
					ModBus.MB_Query.Write_Quantity :=1;
					ModBus.MB_Query.Write_Data[0] := BOOL_TO_WORD(Abilita_UTA12);
					ModBus.MB_Start := TRUE;
					IF 	MB_BitStatoCoil[AddressDaScrivere]=(Abilita_UTA12) THEN
						ScriviRUN_UTA12:=FALSE;
					END_IF
					state := 212;
				ELSE
					state := 212;
				END_IF
			END_IF
		END_IF

		212:    (* Scrittura BOOL Abilita UTA 13 *)
		IF NOT ModBus.MB_Start THEN
			IF ModBus.MB_MASTER.MB_Error<>0 THEN (*OR ModBus.MB_MASTER.MB_Error<>0 THEN*)
				state := 300;
			ELSE
				AddressDaScrivere:=18;
				IF ScriviRUN_UTA13 THEN
					Modbus.MB_Query.FunctionCode := 5;
					Modbus.MB_Query.SlaveAddress := Address;
					ModBus.MB_Query.Write_StartAddress := AddressDaScrivere;
					ModBus.MB_Query.Write_Quantity :=1;
					ModBus.MB_Query.Write_Data[0] := BOOL_TO_WORD(Abilita_UTA13);
					ModBus.MB_Start := TRUE;
					IF 	MB_BitStatoCoil[AddressDaScrivere]=(Abilita_UTA13) THEN
						ScriviRUN_UTA13:=FALSE;
					END_IF
					state := 290;
				ELSE
					state := 290;
				END_IF
			END_IF
		END_IF





		290:    (* Scrittura BOOL - COIL o WORD *)
		IF NOT ModBus.MB_Start THEN
			IF ModBus.MB_MASTER.MB_Error<>0 THEN (*OR ModBus.MB_MASTER.MB_Error<>0 THEN*)
				state := 300;
			ELSE
				IF ScriviDato THEN
					IF ScriviCoil THEN
						Modbus.MB_Query.FunctionCode := 5;
					ELSE
						Modbus.MB_Query.FunctionCode := 6;
					END_IF
					Modbus.MB_Query.SlaveAddress := Address;
					ModBus.MB_Query.Write_StartAddress := IndirizzoDaScrivere;
					ModBus.MB_Query.Write_Quantity :=1;
					ModBus.MB_Query.Write_Data[0] := DatoDaScrivere;
					ModBus.MB_Start := TRUE;
						IF Test_ScriviCoil THEN
							IF 	MB_BitStatoCoil[IndirizzoDaScrivere]=WORD_TO_BOOL(DatoDaScrivere) THEN
								ScriviDato:=FALSE;
							END_IF
						ELSE
							IF 	MB_RegistriHoldingLetti[IndirizzoDaScrivere]=DatoDaScrivere THEN
								ScriviDato:=FALSE;
							END_IF
						END_IF
					state := 295;
				ELSE
					state := 295;
				END_IF
			END_IF
		END_IF



		295:
		IF NOT ModBus.MB_Start THEN
			IF ModBus.MB_MASTER.MB_Error<>0 THEN (*OR ModBus.MB_MASTER.MB_Error<>0 THEN*)
				state := 300;
			ELSE
				IF fModbusAlr THEN fModbusAlr := FALSE; END_IF
				NodoDaInterrogareANZ:=Address+1;
				InibiscoModbusANZ:=FALSE;
				retryErr := 0;
				retry := 0;
				state := 0;
					IF fModbusAlr=FALSE AND ErroreComuModBus=TRUE THEN
						LogEv(EL_Log,EO_CHI,ID,62,'ComunicazioneModBus_OK');
						ErroreComuModBus := FALSE;
				(*	WarningCtr := SEL(WarningCtr=0, WarningCtr-1, 0); *)
					END_IF


			END_IF
		END_IF



	(**** CHECK MODBUS ERROR ****)
	300: 	(* Release MODBUS *)
			InibiscoModbusMB1:=FALSE;
			(* Retries *)
			retry:=retry+1;
			IF retry>3 THEN
				retry:=0;

				(* Verify if slave is dead *)
				IF retryErr < retryErrMaX THEN
					retryErr := retryErr + 1;
				ELSE
					fModbusAlr := TRUE;
					(* Verify ModBus error	*)

					IF fModbusAlr AND ErroreComuModBus=FALSE THEN
						LogEv(EL_Alarm,EO_CHI,ID,61,CONCAT('ErroreModbus_',INT_TO_STRING(ModBus.MB_MASTER.MB_Error)));
						ErroreComuModBus := TRUE;
					END_IF
				END_IF

				END_IF
			Refresh_Now := FALSE;
			InibiscoModbusMB1:=FALSE;
			NodoDaInterrogareMB1:=Address;
			state:=0;
END_CASE




(* Controllo Time Out Ciclo ModBus *)

TimeOutModBus(In:=state<>0,PT:=t#30s);
IF TimeOutModBus.Q THEN
	State:=0;
	Refresh_Now:=TRUE;  (* Rilancio la lettura del nodo *)
	IF MODBUS.MB_Lock=TRUE THEN MODBUS.MB_Lock:=FALSE;END_IF
	IF InibiscoModbusMB1=TRUE THEN InibiscoModbusMB1:=FALSE;END_IF
END_IF
END_ACTION

(* POU Plant_Objects/obj_UTA_02, ST *)
FUNCTION_BLOCK obj_UTA_02
VAR_INPUT
	ID				: BYTE;

	UTA_ST : BOOL;
	UTA_CentrAL : BOOL;
	UTA_AUTO:BOOL:=TRUE;

	(* Physical inputs (Force) *)
	UTA_RUN_REQ		: BOOL; (* External run request (no heat or cold requested) *)
	UTA_STOP_REQ	: BOOL; (* External stop request (has priority over RUN signals!) *)



	cmd_DI_RUN: BOOL;

	T_AMB: INT;
	UR_AMB: INT;
	T_MISC: INT;
	UR_MISC: INT;
	T_MAND: INT;
	T_EST: INT;
	UR_EST: INT;
	ENTALPIA_EST: INT;
	ENTALPIA_AMB: INT;
	UMID_ASS_EST: INT;
	UMID_ASS_AMB: INT;
	UMID_ASS_MISC: INT;
	UMID_ASS_CONDEN: INT;
	SET_COMP_T_AMB: INT;
	RITAR_SET_T_AMB: INT;
	SET_T_MAND: INT;
	SET_ANTIGELO: INT;
	SET_UR_AMB: INT;
	ISTERESI_UR_AMB: INT;
	SET_F_ANTIG_AMB: INT;
	SOGLIA_T_EST_VR: INT;
	MIN_AP_SERR_E_R: INT;
	MIN_AP_SERR_ESP: INT;
	RID_SET_T_RISC: INT;
	VENT_MAND: BOOL;
	VENT_RIPR: BOOL;
	P_UMIDIF: BOOL;
	VALV_B_FREDDA: BOOL;
	VALV_B_CALDA: BOOL;
	SERRANDE_ESP: BOOL;
	SERRAND_EST_RIC: BOOL;
	ABILITA: BOOL;
	STATO_VENT_M: BOOL;
	STATO_VENT_R: BOOL;
	FILTRO: BOOL;
	FLUSSO_VM: BOOL;
	FLUSSO_VR: BOOL;
	FILTRI_INTASATI: BOOL;
	ALL_VERIFICA_VM: BOOL;
	ALL_VERIFICA_VR: BOOL;
	ALL_V011_MANC_SPEGN: BOOL;
	ALL_V011_MANC_FUNZ: BOOL;
	ALL_V012_MANC_SPEGN: BOOL;
	ALL_V012_MANC_FUNZ: BOOL;


END_VAR
VAR_OUTPUT

	cmd_DO_OUT: BOOL;
END_VAR
VAR

	Status_Log		: WORD;
	Status_Vis		: DWORD;


	AllarmeScattoTermico: BOOL;
	AlarmHw		:	FLT_TAP := (INITEV:=FALSE);

(* per creazione stringa da loggare ***)
	temp :STRING(255);
	tempRaw		: ARRAY [0..MAX_SEND_TCP_CLIENT] OF BYTE;
	tempRawLen :DINT;
	longString:STRING(800);



END_VAR
	IF UTA_STOP_REQ THEN cmd_DO_OUT := FALSE;
		ELSIF UTA_RUN_REQ THEN cmd_DO_OUT := TRUE;
		ELSE cmd_DO_OUT := cmd_DI_RUN  ;
	END_IF



(* Hardware alarm (physical input *)
AlarmHw(IN:=UTA_CentrAL);

IF AlarmHw.EVH THEN
	LogEv(EL_Alarm,EO_UTACOIN,ID,3,'UTA_Riarmato');
	AllarmeScattoTermico := FALSE;
END_IF

IF AlarmHw.EVL THEN
	LogEv(EL_Log,EO_UTACOIN,ID,4,'AllarmeUTA');
	AllarmeScattoTermico := TRUE;
END_IF








(* segnalazione Allarme *)
IF AllarmeScattoTermico  THEN
	Status_Log := 2;
	Status_Vis := COLOR_RED;

ELSE
	Status_Log := 0;
	Status_Vis := COLOR_GREEN;
END_IF
END_FUNCTION_BLOCK
ACTION AddLogData:
Logger.s1:=INSERT('&UTACOIN=',BYTE_TO_STRING(ID),8);
IF ID<10 THEN Logger.s1:=INSERT(Logger.s1,'0',8); END_IF


(* inizializzo stringa da loggare **)
FOR tempRawLen:=0 TO MAX_SEND_TCP_CLIENT DO
                tempRaw[tempRawLen]:=0;
END_FOR

tempRawLen:=0;


temp:=Logger.s1;
ADDSTRING(ADR(tempRaw), ADR(temp), tempRawLen);



	temp:=CONCAT(INT_TO_STRING(T_AMB),';');
	ADDSTRING(ADR(tempRaw), ADR(temp), tempRawLen);
	temp:=CONCAT(INT_TO_STRING(UR_AMB),';');
	ADDSTRING(ADR(tempRaw), ADR(temp), tempRawLen);
	temp:=CONCAT(INT_TO_STRING(T_MISC),';');
	ADDSTRING(ADR(tempRaw), ADR(temp), tempRawLen);
	temp:=CONCAT(INT_TO_STRING(UR_MISC),';');
	ADDSTRING(ADR(tempRaw), ADR(temp), tempRawLen);
	temp:=CONCAT(INT_TO_STRING(T_MAND),';');
	ADDSTRING(ADR(tempRaw), ADR(temp), tempRawLen);
	temp:=CONCAT(INT_TO_STRING(T_EST),';');
	ADDSTRING(ADR(tempRaw), ADR(temp), tempRawLen);
	temp:=CONCAT(INT_TO_STRING(UR_EST),';');
	ADDSTRING(ADR(tempRaw), ADR(temp), tempRawLen);
	temp:=CONCAT(INT_TO_STRING(ENTALPIA_EST),';');
	ADDSTRING(ADR(tempRaw), ADR(temp), tempRawLen);
	temp:=CONCAT(INT_TO_STRING(ENTALPIA_AMB),';');
	ADDSTRING(ADR(tempRaw), ADR(temp), tempRawLen);
	temp:=CONCAT(INT_TO_STRING(UMID_ASS_EST),';');
	ADDSTRING(ADR(tempRaw), ADR(temp), tempRawLen);
	temp:=CONCAT(INT_TO_STRING(UMID_ASS_AMB),';');
	ADDSTRING(ADR(tempRaw), ADR(temp), tempRawLen);
	temp:=CONCAT(INT_TO_STRING(UMID_ASS_MISC),';');
	ADDSTRING(ADR(tempRaw), ADR(temp), tempRawLen);
	temp:=CONCAT(INT_TO_STRING(UMID_ASS_CONDEN),';');
	ADDSTRING(ADR(tempRaw), ADR(temp), tempRawLen);
	temp:=CONCAT(INT_TO_STRING(SET_COMP_T_AMB),';');
	ADDSTRING(ADR(tempRaw), ADR(temp), tempRawLen);
	temp:=CONCAT(INT_TO_STRING(RITAR_SET_T_AMB),';');
	ADDSTRING(ADR(tempRaw), ADR(temp), tempRawLen);
	temp:=CONCAT(INT_TO_STRING(SET_T_MAND),';');
	ADDSTRING(ADR(tempRaw), ADR(temp), tempRawLen);
	temp:=CONCAT(INT_TO_STRING(SET_ANTIGELO),';');
	ADDSTRING(ADR(tempRaw), ADR(temp), tempRawLen);
	temp:=CONCAT(INT_TO_STRING(SET_UR_AMB),';');
	ADDSTRING(ADR(tempRaw), ADR(temp), tempRawLen);
	temp:=CONCAT(INT_TO_STRING(ISTERESI_UR_AMB),';');
	ADDSTRING(ADR(tempRaw), ADR(temp), tempRawLen);
	temp:=CONCAT(INT_TO_STRING(SET_F_ANTIG_AMB),';');
	ADDSTRING(ADR(tempRaw), ADR(temp), tempRawLen);
	temp:=CONCAT(INT_TO_STRING(SOGLIA_T_EST_VR),';');
	ADDSTRING(ADR(tempRaw), ADR(temp), tempRawLen);
	temp:=CONCAT(INT_TO_STRING(MIN_AP_SERR_E_R),';');
	ADDSTRING(ADR(tempRaw), ADR(temp), tempRawLen);
	temp:=CONCAT(INT_TO_STRING(MIN_AP_SERR_ESP),';');
	ADDSTRING(ADR(tempRaw), ADR(temp), tempRawLen);
	temp:=CONCAT(INT_TO_STRING(RID_SET_T_RISC),';');
	ADDSTRING(ADR(tempRaw), ADR(temp), tempRawLen);


	temp:=CONCAT(SEL(VENT_MAND,'0','1'),';');
	ADDSTRING(ADR(tempRaw), ADR(temp), tempRawLen);
	temp:=CONCAT(SEL(VENT_RIPR,'0','1'),';');
	ADDSTRING(ADR(tempRaw), ADR(temp), tempRawLen);
	temp:=CONCAT(SEL(P_UMIDIF,'0','1'),';');
	ADDSTRING(ADR(tempRaw), ADR(temp), tempRawLen);
	temp:=CONCAT(SEL(VALV_B_FREDDA,'0','1'),';');
	ADDSTRING(ADR(tempRaw), ADR(temp), tempRawLen);
	temp:=CONCAT(SEL(VALV_B_CALDA,'0','1'),';');
	ADDSTRING(ADR(tempRaw), ADR(temp), tempRawLen);
	temp:=CONCAT(SEL(SERRANDE_ESP,'0','1'),';');
	ADDSTRING(ADR(tempRaw), ADR(temp), tempRawLen);
	temp:=CONCAT(SEL(SERRAND_EST_RIC,'0','1'),';');
	ADDSTRING(ADR(tempRaw), ADR(temp), tempRawLen);
	temp:=CONCAT(SEL(ABILITA,'0','1'),';');
	ADDSTRING(ADR(tempRaw), ADR(temp), tempRawLen);
	temp:=CONCAT(SEL(STATO_VENT_M,'0','1'),';');
	ADDSTRING(ADR(tempRaw), ADR(temp), tempRawLen);
	temp:=CONCAT(SEL(STATO_VENT_R,'0','1'),';');
	ADDSTRING(ADR(tempRaw), ADR(temp), tempRawLen);
	temp:=CONCAT(SEL(FILTRO,'0','1'),';');
	ADDSTRING(ADR(tempRaw), ADR(temp), tempRawLen);
	temp:=CONCAT(SEL(FLUSSO_VM,'0','1'),';');
	ADDSTRING(ADR(tempRaw), ADR(temp), tempRawLen);
	temp:=CONCAT(SEL(FLUSSO_VR,'0','1'),';');
	ADDSTRING(ADR(tempRaw), ADR(temp), tempRawLen);
	temp:=CONCAT(SEL(FILTRI_INTASATI,'0','1'),';');
	ADDSTRING(ADR(tempRaw), ADR(temp), tempRawLen);
	temp:=CONCAT(SEL(ALL_VERIFICA_VM,'0','1'),';');
	ADDSTRING(ADR(tempRaw), ADR(temp), tempRawLen);
	temp:=CONCAT(SEL(ALL_VERIFICA_VR,'0','1'),';');
	ADDSTRING(ADR(tempRaw), ADR(temp), tempRawLen);
	temp:=CONCAT(SEL(ALL_V011_MANC_SPEGN,'0','1'),';');
	ADDSTRING(ADR(tempRaw), ADR(temp), tempRawLen);
	temp:=CONCAT(SEL(ALL_V011_MANC_FUNZ,'0','1'),';');
	ADDSTRING(ADR(tempRaw), ADR(temp), tempRawLen);
	temp:=CONCAT(SEL(ALL_V012_MANC_SPEGN,'0','1'),';');
	ADDSTRING(ADR(tempRaw), ADR(temp), tempRawLen);
	temp:=SEL(ALL_V012_MANC_FUNZ,'0','1');
	ADDSTRING(ADR(tempRaw), ADR(temp), tempRawLen);


ADDSTRING(ADR(Logger.TData), ADR(tempRaw), Logger.TLen);


(*



Logger.s1:=CONCAT(Logger.s1,SEL(UTA_ST,'0','100'));		Logger.s1:=CONCAT(Logger.s1,';');

Logger.s1:=CONCAT(Logger.s1,WORD_TO_STRING(Status_Log));
Logger.s1:=CONCAT(Logger.s1,';');
Logger.s1:=CONCAT(Logger.s1,SEL(UTA_RUN_REQ,'0','100'));
Logger.s1:=CONCAT(Logger.s1,';');
Logger.s1:=CONCAT(Logger.s1,SEL(UTA_STOP_REQ,'0','100'));

Logger.s1:=CONCAT(Logger.s1,';');
Logger.s1:=CONCAT(Logger.s1,SEL(UTA_AUTO,'1','0'));


ADDSTRING(ADR(Logger.TData), ADR(Logger.s1), Logger.TLen);

*)
END_ACTION

(* POU Plant_Objects/obj_ZTHL_01, ST *)
FUNCTION_BLOCK obj_ZTHL_01
(* === ZIGBEE AMBIENT SENSORS MT-200 ===
   v1.0[07/05/05] - Create
*)
VAR CONSTANT
	LQI_Threshold		:	WORD := 10;		(* Zigbee link quality minimum value *)
	LowBattVoltage		:	WORD := 2700;		(* Battery is considered low when reaches 1.35V each *)
END_VAR
VAR_INPUT
	(* Settings *)
	ID				: BYTE;
	Address			: BYTE;

(*	Refresh_Period	: TIME:=t#5m;
	(* Controls *)
	Refresh_Auto	: BOOL:=TRUE; (* Enable automatic refresh *)*)

	(* Modbus *)
	Refresh_Now	:	BOOL;	(* Start immediately modbus state machine *)
	retryErrMax	:	BYTE := 2;

	(* Limits *)
	Tmin			: INT := 50;
	Tmax			: INT := 400;
END_VAR
VAR_IN_OUT
	(* Interface *)
	ModBus		:obj_MODBUS;

END_VAR
VAR_OUTPUT
	(* Status *)
	Status_Log		: BYTE;
	Status_Vis 		: DWORD;
END_VAR
VAR


	state		:	INT;
	retry		:	BYTE;
	retryErr	:	BYTE;
	ReadTmr		:	TON := (PT:=T#5s);
	fModbusAlr:BOOL;


	AlarmCtr		: BYTE;
	WarningCtr		: BYTE;

	id_locale: BYTE;

	MB_RegistriLetti: ARRAY [0..20] OF INT;

	Quality			: FLT_EVENT;
	Battery			: FLT_EVENT;
	Temperature		: FLT_EVENT := (INITEV:=FALSE);
	Alarm			: FLT_EVENT;

	ERR				: BOOL;
	fLQI			: BOOL;
	fBatt			: BOOL;
	fTemp			: BOOL;

	StatusOK		: BYTE;			(* 0: Status OK, >=1: Alarm and/or warning		Incremented by 1 when Alarm or Wrn occurs,
																					decremented by 1 when restored	*)
	TimeOutModBus: TON;
	ErroreComuModBus: BOOL;

	VerificaFuctionCode: INT;
	VerificaNodoLetto: INT;


END_VAR
(* stato creato per potere interrogare il nodo corretto *)
id_locale:=ID;

Stm();

checkAlarm();
END_FUNCTION_BLOCK
ACTION AddLogData:
Logger.s1:=INSERT('&ZTHL=',BYTE_TO_STRING(ID),5);
IF ID<10 THEN Logger.s1:=INSERT(Logger.s1,'0',5); END_IF

Logger.s1:=CONCAT(Logger.s1,INT_TO_STRING(MB_RegistriLetti[3]));	(* Livello segnale radio dell'ultimo messaggio ricevuto dal dispositivo  *)
Logger.s1:=CONCAT(Logger.s1,';');
Logger.s1:=CONCAT(Logger.s1,INT_TO_STRING(MB_RegistriLetti[6]));	(* Temperatura (in decimi di grado centigrado)  *)
Logger.s1:=CONCAT(Logger.s1,';');
Logger.s1:=CONCAT(Logger.s1,INT_TO_STRING(MB_RegistriLetti[8]));	(* Umidità (espressa in % Umidità Relativa)  *)
Logger.s1:=CONCAT(Logger.s1,';');
Logger.s1:=CONCAT(Logger.s1,INT_TO_STRING(MB_RegistriLetti[5]));	(* Valore efficace Luce (espressa in Lux)  *)
Logger.s1:=CONCAT(Logger.s1,';');
Logger.s1:=CONCAT(Logger.s1,INT_TO_STRING(MB_RegistriLetti[4]));	(* Livello di Batteria (in millesimi di volt) *)
Logger.s1:=CONCAT(Logger.s1,';');

Logger.s1:=CONCAT(Logger.s1,BYTE_TO_STRING(Status_Log));
ADDSTRING(ADR(Logger.TData), ADR(Logger.s1), Logger.TLen);
END_ACTION
ACTION CheckAlarm:
(**** GEstione Log ad Evento *****)


(* (MB_RegistriLetti[3]) check Livello segnale radio dell'ultimo messaggio ricevuto dal dispositivo *)

IF (MB_RegistriLetti[3]) < LQI_Threshold THEN
	fLQI := FALSE;
	ERR := TRUE;
ELSE
	fLQI := TRUE;
	ERR := FALSE;
END_IF

Quality(IN:=fLQI);

IF Quality.EVL THEN
	LogEv(SEL((MB_RegistriLetti[3])<>0,EL_Alarm,EL_Wrn),EO_ZTHL,ID,SEL((MB_RegistriLetti[3])<>0,7,2),WORD_TO_STRING((MB_RegistriLetti[3])));
	Status_Log := SEL((MB_RegistriLetti[3])<>0,2,1);
	StatusOK := StatusOK + 1;
END_IF

IF Quality.EVH THEN StatusOK := SEL(StatusOK=0, StatusOK-1, 0); END_IF

(* If probe (node) is present proceed checking other warnings, otherwise don't transmit anything *)
IF (MB_RegistriLetti[3]) <> 0 THEN

	(* Check battery voltage *)

(* (MB_RegistriLetti[4]) check Livello di Batteria (in millesimi di volt) *)

	IF (MB_RegistriLetti[4]) < LowBattVoltage THEN fBatt := TRUE;
	ELSE fBatt := FALSE;
	END_IF


	Battery(IN:=fBatt);

	IF Battery.EVH  THEN
		LogEv(EL_Wrn,EO_ZTHL,ID,6,' ');
		StatusOK := StatusOK + 1;
	END_IF

	IF Battery.EVL THEN StatusOK := SEL(StatusOK=0, StatusOK-1, 0); END_IF

(* (MB_RegistriLetti[6]) check Temperatura (in decimi di grado centigrado) *)

	(* Check Node temperature *)
	IF (MB_RegistriLetti[6]) < Tmin OR (MB_RegistriLetti[6]) > Tmax THEN
		fTemp := TRUE;
		ERR := TRUE;
	ELSE
		fTemp := FALSE;
		ERR := FALSE;
	END_IF

	Temperature(IN:=fTemp);

	IF Temperature.EVH THEN
		LogEv(EL_Wrn,EO_ZTHL,ID,5,INT_TO_STRING((MB_RegistriLetti[6])));
		Status_Log := 1;
		StatusOK := StatusOK + 1;
	END_IF

	IF Temperature.EVL THEN StatusOK := SEL(StatusOK=0, StatusOK-1, 0); END_IF

END_IF

Alarm(IN:=(StatusOK=0));

IF Alarm.EVH THEN
	Status_Log := 0;
	LogEv(EL_Log,EO_ZTHL,ID,1,'');
END_IF

IF Status_Log = 2 THEN Status_Vis := COLOR_RED;
ELSIF Status_Log = 1 THEN Status_Vis := COLOR_YELLOW;
ELSE Status_Vis := COLOR_GREEN;
END_IF
END_ACTION
ACTION Stm:
CASE state OF
	0:	(* Refresh time manager *)
		ReadTmr(IN:=NOT ReadTmr.Q);
		(*A tempo interrogo il nodo sempre che non ci sia qualcuno che lo sta interrogando in quel momento *)

		IF (ReadTmr.Q AND NodoDaInterrogareMB2=id_locale )OR Refresh_Now AND NOT InibiscoModbusMB2 THEN
			state := 10;
			ReadTmr.PT := T#5s;  (* moreno *)
			Refresh_Now := FALSE;
			InibiscoModbusMB2 := TRUE;
		END_IF

	(**** Leggo le Analogiche a Disposzione  ****)

	10:	(* richiedo lettura Holding Register   *)

		Modbus.MB_Query.SlaveAddress := Address;
		Modbus.MB_Query.FunctionCode := 4;
		ModBus.MB_Query.Read_StartAddress := 0 ;			(* richiedo lettura altri Parametri *)
		ModBus.MB_Query.Read_Quantity := 10;
		ModBus.MB_Start := TRUE;
		state := 20;

	20:	(* Risposta all'interrogazione *)
		IF NOT ModBus.MB_Start   THEN
			VerificaFuctionCode:=ModBus.MB_Resp.FunctionCode;
			VerificaNodoLetto:=ModBus.MB_Resp.SlaveAddress;

			IF ModBus.MB_MASTER.MB_Error<>0 THEN
				state := 300;
			ELSE

				MB_RegistriLetti[0] := ModBus.MB_Resp.Data[0];   	(* Vedi tabella *)
				MB_RegistriLetti[1] := ModBus.MB_Resp.Data[1];		(* Vedi tabella *)
				MB_RegistriLetti[2] := ModBus.MB_Resp.Data[2];		(* Vedi tabella *)
				MB_RegistriLetti[3] := ModBus.MB_Resp.Data[3];		(* Vedi tabella *)
				MB_RegistriLetti[4] := ModBus.MB_Resp.Data[4];		(* Vedi tabella *)
				MB_RegistriLetti[5] := ModBus.MB_Resp.Data[5];		(* Vedi tabella *)
				MB_RegistriLetti[6] := ModBus.MB_Resp.Data[6];		(* Vedi tabella *)
				MB_RegistriLetti[7] := ModBus.MB_Resp.Data[7];		(* Vedi tabella *)
				MB_RegistriLetti[8] := ModBus.MB_Resp.Data[8];		(* Vedi tabella *)
				MB_RegistriLetti[9] := ModBus.MB_Resp.Data[9];		(* Vedi tabella *)
				MB_RegistriLetti[10] := ModBus.MB_Resp.Data[10];		(* Vedi tabella *)
				MB_RegistriLetti[11] := ModBus.MB_Resp.Data[11];		(* Vedi tabella *)
				MB_RegistriLetti[12] := ModBus.MB_Resp.Data[12];		(* Vedi tabella *)
				MB_RegistriLetti[13] := ModBus.MB_Resp.Data[13];		(* Vedi tabella *)

				state := 295;
			END_IF
		END_IF


		295:
		IF NOT ModBus.MB_Start THEN
			IF ModBus.MB_MASTER.MB_Error<>0 THEN (*OR ModBus.MB_MASTER.MB_Error<>0 THEN*)
				state := 300;
			ELSE
				IF fModbusAlr THEN fModbusAlr := FALSE; END_IF
				NodoDaInterrogareMB2:=id_locale+1;
				InibiscoModbusMB2:=FALSE;
				retryErr := 0;
				retry := 0;
				state := 0;
					IF fModbusAlr=FALSE AND ErroreComuModBus=TRUE THEN
						LogEv(EL_Log,EO_CHI,ID,62,'ComunicazioneModBus_OK');
						ErroreComuModBus := FALSE;
				(*	WarningCtr := SEL(WarningCtr=0, WarningCtr-1, 0); *)
					END_IF


			END_IF
		END_IF



	(**** CHECK MODBUS ERROR ****)
	300: 	(* Release MODBUS *)
			InibiscoModbusMB3:=FALSE;
			(* Retries *)
			retry:=retry+1;
			IF retry>3 THEN
				retry:=0;

				(* Verify if slave is dead *)
				IF retryErr < retryErrMaX THEN
					retryErr := retryErr + 1;
				ELSE
					fModbusAlr := TRUE;
					(* Verify ModBus error	*)

					IF fModbusAlr AND ErroreComuModBus=FALSE THEN
						LogEv(EL_Alarm,EO_CHI,ID,61,CONCAT('ErroreModbus_',INT_TO_STRING(ModBus.MB_MASTER.MB_Error)));
						ErroreComuModBus := TRUE;
					END_IF
				END_IF

			END_IF
			Refresh_Now := FALSE;
			InibiscoModbusMB2:=FALSE;
			NodoDaInterrogareMB2:=id_locale+1;
			state:=0;
END_CASE




(* Controllo Time Out Ciclo ModBus *)

TimeOutModBus(In:=state<>0,PT:=t#30s);
IF TimeOutModBus.Q THEN
	State:=0;
	Refresh_Now:=TRUE;  (* Rilancio la lettura del nodo *)
	IF MODBUS.MB_Lock=TRUE THEN MODBUS.MB_Lock:=FALSE;END_IF
	IF InibiscoModbusMB2=TRUE THEN InibiscoModbusMB2:=FALSE;END_IF
END_IF
END_ACTION

(* POU Utils Functions/PLANT_STATUS, ST *)
FUNCTION_BLOCK PLANT_STATUS
VAR_INPUT
	obj_Status		:	WORD;
END_VAR
VAR_OUTPUT
END_VAR
VAR
	PLANT_STATUS	:	WORD;

	Pwm				:	TON := (PT:=T#1s);
END_VAR
CASE plant_Status OF

	0:	(* Plant OK - Everything works well *)
		(*Pwm(IN:=FALSE);	*)						(* Stop timer if running *)
		LAMP_AL := FALSE;						(* Keep the lamp switched off *)

	(*1:	(* Plant in warning *)
		Pwm(IN:= NOT(Pwm.Q));

		IF Pwm.Q THEN
			LAMP_AL := NOT LAMP_AL;				(* Toggle output *)
		END_IF*)

	2:	(* Plant in alarm *)
		(*Pwm(IN:=FALSE);	*)						(* Stop timer if running *)
		LAMP_AL	:= TRUE;						(* Keep the lamp switched on *)

END_CASE

plant_Status := 0;		(* Reset plant status *)
END_FUNCTION_BLOCK
ACTION UpdateStatus:
IF plant_Status = 2 THEN

	RETURN;					(* If plant already in alarm condition do nothing *)

ELSE

		IF obj_Status <> 0 THEN
			plant_Status := obj_Status;			(* If plant in warning/normal condition and current object in alarm, update plant status *)
		END_IF
END_IF
END_ACTION

(* POU PLC_WDT, ST *)
FUNCTION PLC_WDT: DWORD VAR_INPUT dwEvent: DWORD; dwFilter: DWORD; dwOwner: DWORD; END_VAR
LogEv(EL_AlarmStop,EO_SYS,1,10,'Watchdog');
END_FUNCTION

(* POU Utils Functions/RAW16TOHEXSTR, ST *)
FUNCTION RAW16TOHEXSTR : STRING(128)
VAR_INPUT
	pData: POINTER TO BYTE;
	DataLen: BYTE;
END_VAR
VAR
	pt: POINTER TO BYTE;
	xl: BYTE;
END_VAR
pt:=ADR(RAW16TOHEXSTR);
xl:=0;

WHILE DataLen>0 AND xl<120 DO

	pData:=pData+1;

	pt^ := (pData^ / 16#10) + 48 + (((pData^ / 16#10)/10)*7);
	pt:=pt+1;
	pt^ := (pData^ AND 16#0F)  + 48 + (((pData^ AND 16#0F)/10)*7);
	pt:=pt+1;

	pData:=pData-1;

	pt^ := (pData^ / 16#10) + 48 + (((pData^ / 16#10)/10)*7);
	pt:=pt+1;
	pt^ := (pData^ AND 16#0F)  + 48 + (((pData^ AND 16#0F)/10)*7);
	pt:=pt+1;

	xl:=xl+4;

	DataLen:=DataLen-2;
	pData:=pData+2;

END_WHILE

pt^:=0;
END_FUNCTION

(* POU Utils Functions/RAWTOHEXSTR, ST *)
FUNCTION RAWTOHEXSTR : STRING(128)
VAR_INPUT
	pData: POINTER TO BYTE;
	DataLen: BYTE;
END_VAR
VAR
	pt: POINTER TO BYTE;
	xl: BYTE;
END_VAR
pt:=ADR(RAWTOHEXSTR);

xl:=2;

WHILE DataLen>0 AND xl<128 DO

	pt^ := (pData^ / 16#10) + 48 + (((pData^ / 16#10)/10)*7);
	pt:=pt+1;
	pt^ := (pData^ AND 16#0F)  + 48 + (((pData^ AND 16#0F)/10)*7);
	pt:=pt+1;

	xl:=xl+2;

	DataLen:=DataLen-1;
	pData:=pData+1;

END_WHILE

pt^:=0;
END_FUNCTION

(* POU Utils/RTC_Update, ST *)
FUNCTION RTC_Update : BOOL
VAR
	T: DT;
	TS: STRING;
	TS2: STRING;
	Hour: BYTE;
	Minute: BYTE;
END_VAR
(* Get RTC time *)
T:=SysRtcGetTime(TRUE);
Sys.Time_CT_DT:=T;
(* Calculate variables *)
TS:=DT_TO_STRING(T);
Sys.Time_LogString:=DELETE(STR:=TS, LEN:=3, POS:=1);
TS2:=MID(STR:=TS, LEN:=4, POS:= 4); Sys.Time_Year 	:=STRING_TO_WORD(TS2);
TS2:=MID(STR:=TS, LEN:=2, POS:= 9); Sys.Time_Month	:=STRING_TO_BYTE(TS2);
TS2:=MID(STR:=TS, LEN:=2, POS:=12); Sys.Time_Day  	:=STRING_TO_BYTE(TS2);
Sys.Time_CT_Day:=(32*(Sys.Time_Month-1)+Sys.Time_Day-1);
TS2:=MID(STR:=TS, LEN:=2, POS:=15); Hour			:=STRING_TO_BYTE(TS2);
TS2:=MID(STR:=TS, LEN:=2, POS:=18); Minute		 	:=STRING_TO_BYTE(TS2);
Sys.Time_Hour := Hour;
Sys.Time_Minute := Minute;
Sys.Time_CT_Quarter:=Hour*4+(Minute/15);
END_FUNCTION

(* POU Utils Functions/SHIFT_ARRAY, ST *)
FUNCTION SHIFT_ARRAY : BOOL
VAR_INPUT
	pData	:	POINTER TO ARRAY [1..2] OF WORD;
	Size	:	BYTE;
END_VAR
VAR
	pNew	:	POINTER TO WORD;
	i		:	BYTE;
END_VAR
(* Shift right *)
FOR i:=1 TO (Size-1) BY 1 DO

	(*pNew := pData + 1;*)
	pData^[i] := pData^[i+1];
	(*pData := pData + 1;*)

END_FOR
END_FUNCTION

(* Visualisation PLC_VISU
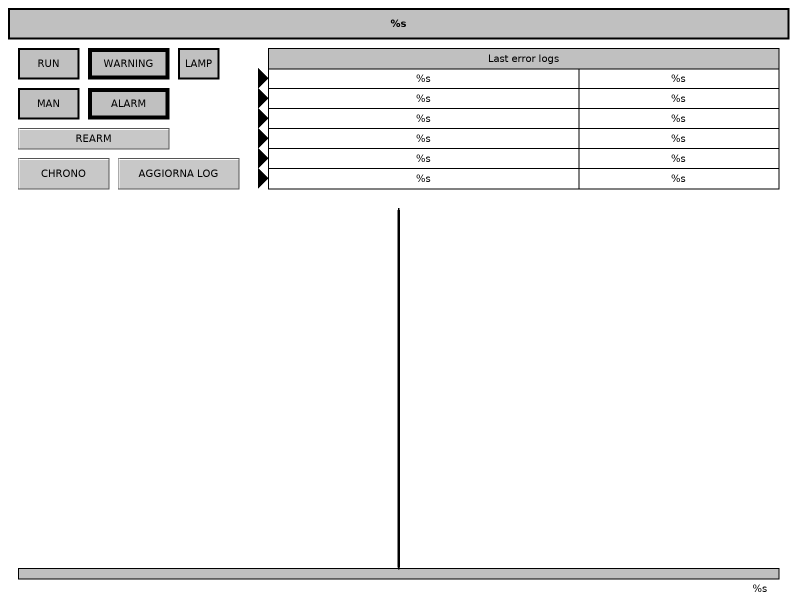
rectangle at (10,10)-(791,41): text "%s"; shows .Plant_NAME
rectangle at (530,580)-(771,601): text "%s"; shows Sys.Time_LogString
rounded rectangle at (20,50)-(81,81): text "RUN"; alarm colour if NOT Mode_Manual; runs INTERN ASSIGN Mode_Manual:=(FALSE)
rounded rectangle at (20,90)-(81,121): text "MAN"; alarm colour if Mode_Manual; runs INTERN ASSIGN Mode_Manual:=(TRUE)
rectangle at (580,70)-(781,91): text "%s"; shows Sys.LastLogs_Msg[0]
polygon at (260,170)-(270,190): invisible if Sys.LastLogs_Idx<>0
rectangle at (580,90)-(781,111): text "%s"; shows Sys.LastLogs_Msg[1]
polygon at (260,70)-(270,90): invisible if Sys.LastLogs_Idx<>1
rectangle at (580,110)-(781,131): text "%s"; shows Sys.LastLogs_Msg[2]
polygon at (260,90)-(270,110): invisible if Sys.LastLogs_Idx<>2
rectangle at (580,130)-(781,151): text "%s"; shows Sys.LastLogs_Msg[3]
polygon at (260,110)-(270,130): invisible if Sys.LastLogs_Idx<>3
rectangle at (580,150)-(781,171): text "%s"; shows Sys.LastLogs_Msg[4]
polygon at (260,130)-(270,150): invisible if Sys.LastLogs_Idx<>4
rectangle at (580,170)-(781,191): text "%s"; shows Sys.LastLogs_Msg[5]
polygon at (260,150)-(270,170): invisible if Sys.LastLogs_Idx<>5
rectangle at (270,70)-(581,91): text "%s"; shows Sys.LastLogs_Dat[0]
rectangle at (270,90)-(581,111): text "%s"; shows Sys.LastLogs_Dat[1]
rectangle at (270,110)-(581,131): text "%s"; shows Sys.LastLogs_Dat[2]
rectangle at (270,130)-(581,151): text "%s"; shows Sys.LastLogs_Dat[3]
rectangle at (270,150)-(581,171): text "%s"; shows Sys.LastLogs_Dat[4]
rectangle at (270,170)-(581,191): text "%s"; shows Sys.LastLogs_Dat[5]
rectangle at (90,90)-(171,121): text "ALARM"; alarm colour if Sys.Alarm; runs INTERN ASSIGN Mode_Manual:=(FALSE)
rectangle at (90,50)-(171,81): text "WARNING"; alarm colour if Sys.Warning; runs INTERN ASSIGN Mode_Manual:=(TRUE)
button at (20,130)-(171,151): text "REARM"; runs INTERN ASSIGN Sys.Alarm:=(FALSE);INTERN ASSIGN Sys.Warning:=(FALSE)
rectangle at (270,50)-(781,71): text "Last error logs"
rounded rectangle at (180,50)-(221,81): text "LAMP"; alarm colour if LAMP_AL
button at (20,160)-(111,191): text "CHRONO"; opens VIS_CHONOEDITOR
button at (120,160)-(241,191): text "AGGIORNA LOG"; taps .AggiornaLog
2 more shapes without text or variables
*)

